// TwinCAT 3 PLC project TwinCAT_OpenFramework_Automation
// Title: TwinCAT Open Framework Automation
// Company: Oleksandr Tiutyk FOP
// Author: Oleksandr Tiutyk
// ProjectVersion: 1.0.13.0
// Description: TwinCAT.OpenFramework automation core types and device abstractions
// ProgramVersion: 3.1.4026.28
// libraries:
//   Tc2_Standard, * (Beckhoff Automation GmbH)
//   Tc2_System, * (Beckhoff Automation GmbH)
//   [TwinCAT Open Framework Core], * (Oleksandr Tiutyk FOP)
// project tree:
//   AutomationComponent/Branches/AutomationController/ AutomationController.TcPOU, AutomationControllers.TcPOU, IAutomationController.TcIO
//   AutomationComponent/Branches/AutomationController/Plugins/HMI/ HmiAutomationComponentElement.TcPOU, HMI_AUTOMATION_COMPONENT_COMMANDS.TcDUT, HMI_AUTOMATION_COMPONENT_STATUSES.TcDUT
//   AutomationComponent/Branches/AutomationController/Plugins/ IAutomationControllerPlugin.TcIO
//   AutomationComponent/Branches/ BranchAutomationComponent.TcPOU
//   AutomationComponent/Branches/Composite/ CompositeAutomationComponent.TcPOU, ICompositeAutomationComponent.TcIO
//   AutomationComponent/Branches/ChildCriticalErrorHandlingPolicies/ ChildCriticalErrorHandlingPolicies.TcPOU, CHILD_CRITICAL_ERROR_REACTION.TcDUT, IChildCriticalErrorHandlingPolicy.TcIO, IgnoreChildCriticalErrorHandlingPolicy.TcPOU, SetErrorAndContinueAfterChildCriticalErrorHandlingPolicy.TcPOU, SetErrorAndStopAfterCriticalChildErrorHandlingPolicy.TcPOU
//   AutomationComponent/Enums/ OPERATIONAL_STATE.TcDUT
//   AutomationComponent/ AutomationComponent.TcPOU, IAutomationComponent.TcIO
//   AutomationComponent/CommonSubInterfaces/ IChildAutomationComponent.TcIO, IInputLeafAutomationComponent.TcIO, IOutputLeafAutomationComponent.TcIO, IParentAutomationComponent.TcIO
//   AutomationComponent/Leafs/InputOutput/ InputOutputLeafAutomationComponent.TcPOU
//   AutomationComponent/Leafs/Input/ InputLeafAutomationComponent.TcPOU
//   AutomationComponent/Leafs/Output/ OutputLeafAutomationComponent.TcPOU
//   AutomationComponent/Leafs/ LeafAutomationComponent.TcPOU
//   AutomationRunner/ AutomationRunner.TcPOU, AUTOMATION_RUNNER_STATE.TcDUT, IAutomationRunner.TcIO
//   Internal/ CurrentNamespace.TcPOU, NamespaceExtractor.TcPOU
//   / Parameters.TcGVL
//   Simulatable/ IChildConfigurableSimulatable.TcIO, IChildSimulatable.TcIO, IConfigurableSimulatable.TcIO, ISimulatable.TcIO, SIMULATION_MODE_OVERRIDE.TcDUT
//   Version/ Global_Version.TcGVL
// (motion and I/O tree: see PLC project twincat_openframework_core)
// real-time tasks:
//   TASK PlcTask: cycle T#10ms, priority 20, ADS port 350
//   TASK TestTask: cycle T#10ms, priority 1, ADS port 351
//   TASK RunnerTestTask: cycle T#10ms, priority 2, ADS port 354
//   TASK HowToTask: cycle T#10ms, priority 22, ADS port 353
// variable links:

// ---- AutomationComponent/Branches/AutomationController/Plugins/HMI/HMI_AUTOMATION_COMPONENT_COMMANDS.TcDUT
(*
SPDX-FileCopyrightText: Â© 2026 Oleksandr Tiutyk <trofimich@gmail.com>
SPDX-License-Identifier: MIT
License: https://opensource.org/license/mit
*)

(*!
<summary>Defines command flags sent from an HMI to an automation component.</summary>
<description>
Command fields are pulsed or set by an operator/HMI interface. The element consumes and resets these flags to FALSE
within its local instance memory upon dispatching the operation.
</description>
*)

TYPE HMI_AUTOMATION_COMPONENT_COMMANDS :
STRUCT
	Enable : BOOL;
	Disable : BOOL;
	
	Reset : BOOL;	
END_STRUCT
END_TYPE

// ---- AutomationComponent/Branches/AutomationController/Plugins/HMI/HMI_AUTOMATION_COMPONENT_STATUSES.TcDUT
(*
SPDX-FileCopyrightText: Â© 2026 Oleksandr Tiutyk <trofimich@gmail.com>
SPDX-License-Identifier: MIT
License: https://opensource.org/license/mit
*)

(*!
<summary>Provides automation component operational state and diagnostics to an HMI.</summary>
<description>
Aggregates enablement, error details, and current operational state information for UI visualization.
</description>
*)

TYPE HMI_AUTOMATION_COMPONENT_STATUSES :
STRUCT
	Enabled : BOOL;

	HasError : BOOL;
	ErrorMessage : TOF_Core.ERROR_MESSAGE;
	ErrorSource : STRING(255);
	ErrorLocalTimestamp : LDATE_AND_TIME;
	ErrorUtcTimestamp : LDATE_AND_TIME;

	OperationalState : OPERATIONAL_STATE;
	OperationalStateName : STRING;
	OperationalStateReason : WSTRING(255);
END_STRUCT
END_TYPE

// ---- AutomationComponent/Branches/ChildCriticalErrorHandlingPolicies/CHILD_CRITICAL_ERROR_REACTION.TcDUT
(*
SPDX-FileCopyrightText: Â© 2026 Oleksandr Tiutyk <trofimich@gmail.com>
SPDX-License-Identifier: MIT
License: https://opensource.org/license/mit
*)

(*!
<summary>Defines reactions for handling critical errors reported by child components.</summary>
<description>
Returned by IChildCriticalErrorHandlingPolicy implementations to determine whether the parent component
should stop execution, continue running with an error state, or ignore the child failure.
</description>
*)

{attribute 'qualified_only'}
{attribute 'to_string'}
TYPE CHILD_CRITICAL_ERROR_REACTION :
(
	(*! <summary>Transition parent into error state and trigger component stop.</summary> *)
	SET_ERROR_AND_STOP,
	(*! <summary>Transition parent into error state but continue cyclic execution.</summary> *)
	SET_ERROR_AND_CONTINUE,
	(*! <summary>Ignore child error and take no action on parent component.</summary> *)
	IGNORE
);
END_TYPE

// ---- AutomationComponent/Enums/OPERATIONAL_STATE.TcDUT
(*
SPDX-FileCopyrightText: © 2026 Oleksandr Tiutyk <trofimich@gmail.com>
SPDX-License-Identifier: MIT
License: https://opensource.org/license/mit
*)

(*!
<summary>Defines the operational lifecycle states of an automation component.</summary>
*)

{attribute 'qualified_only'}
{attribute 'strict'}
{attribute 'to_string'}
TYPE OPERATIONAL_STATE :
(
	INITIALIZING := 0, (*!<description>Start state for self and children initialization.</description>*)
	WORKING,           (*!<description>Normal working mode after successful initialization.</description>*)
	(*!
	<description>
	Recoverable stopped state. Entered after Stop or critical runtime error. Reset required to return to WORKING.
	</description>
	*)
	STOPPED,
	INVALID            (*!<description>Any error occurred during initialization, final state.</description>*)
);
END_TYPE

// ---- AutomationRunner/AUTOMATION_RUNNER_STATE.TcDUT
(*
SPDX-FileCopyrightText: © 2026 Oleksandr Tiutyk <trofimich@gmail.com>
SPDX-License-Identifier: MIT
License: https://opensource.org/license/mit
*)

(*!
<summary>Defines the execution states of an automation runner.</summary>
*)

{attribute 'qualified_only'}
{attribute 'strict'}
{attribute 'to_string'}
TYPE AUTOMATION_RUNNER_STATE :
(
	INITIALIZING := 0, (*!<description>Start state, active until all components complete initialization.</description>*)
	RUNNING := 1,      (*!<description>Normal cyclic execution of automation components.</description>*)
	INVALID := 2       (*!<description>Any fatal initialization error occurred; runner execution halted.</description>*)
);
END_TYPE

// ---- Simulatable/SIMULATION_MODE_OVERRIDE.TcDUT
(*
SPDX-FileCopyrightText: Â© 2026 Oleksandr Tiutyk <trofimich@gmail.com>
SPDX-License-Identifier: MIT
License: https://opensource.org/license/mit
*)

(*!
<summary>Defines simulation mode override behavior for child components.</summary>
<description>
Allows individual child components to follow the parent's simulation state or explicitly force simulation ON or OFF.
</description>
*)

{attribute 'qualified_only'}
{attribute 'strict'}
{attribute 'to_string'}
TYPE SIMULATION_MODE_OVERRIDE :
(
	(*! <summary>Inherit simulation mode from parent component.</summary> *)
	INHERITED := 0,
	(*! <summary>Force simulation mode ON regardless of parent setting.</summary> *)
	ON,
	(*! <summary>Force simulation mode OFF regardless of parent setting.</summary> *)
	OFF
);
END_TYPE

// ---- Parameters.TcGVL
(*
SPDX-FileCopyrightText: Â© 2026 Oleksandr Tiutyk <trofimich@gmail.com>
SPDX-License-Identifier: MIT
License: https://opensource.org/license/mit
*)

(*!
<summary>Defines global configuration parameters for the automation framework.</summary>
*)

{attribute 'qualified_only'}
VAR_GLOBAL CONSTANT
	(*! <summary>Default timeout duration for component initialization phase (5 seconds).</summary> *)
	InitializationTimeout : TIME := T#5S;
END_VAR

// ---- Version/Global_Version.TcGVL
{attribute 'TcGenerated'}
{attribute 'no-analysis'}
{attribute 'linkalways'}
// This function has been automatically generated from the project information.
VAR_GLOBAL CONSTANT
	{attribute 'const_non_replaced'}
	stLibVersion_TwinCAT_Open_Framework_Automation : ST_LibVersion := (iMajor := 1, iMinor := 0, iBuild := 13, iRevision := 0, nFlags := 0, sVersion := '1.0.13.0');
END_VAR

// ---- AutomationComponent/Branches/AutomationController/IAutomationController.TcIO
(*
SPDX-FileCopyrightText: © 2026 Oleksandr Tiutyk <trofimich@gmail.com>
SPDX-License-Identifier: MIT
License: https://opensource.org/license/mit
*)

(*!
<summary>
Defines the root automation controller capable of coordinating child components and controller plugins.
</summary>
<description>Indexed Try lookups return borrowed interfaces or null and do not propagate exceptions.</description>
*)

INTERFACE IAutomationController EXTENDS IParentAutomationComponent

{attribute 'monitoring' := 'call'}
PROPERTY FINAL PluginCount : TOF_Core.INT_LENGTH
GET
END_GET
END_PROPERTY

(*!
<summary>Returns a borrowed plugin by its zero-based index.</summary>
<description>
Returns null when the entry is unavailable, the index is out of range or a nested call raises an exception.
Fatal allocation observations return null and leave the fatal latch set for the outer task boundary.
Does not transfer ownership or extend lifetime. Implementations must not propagate exceptions.
</description>
*)
METHOD TryGetPluginByIndex : IAutomationControllerPlugin
VAR_INPUT
	index : TOF_Core.INT_INDEX;
END_VAR
END_METHOD

END_INTERFACE

// ---- AutomationComponent/Branches/AutomationController/Plugins/IAutomationControllerPlugin.TcIO
(*
SPDX-FileCopyrightText: Â© 2026 Oleksandr Tiutyk <trofimich@gmail.com>
SPDX-License-Identifier: MIT
License: https://opensource.org/license/mit
*)

(*!
<summary>Defines lifecycle extension hooks for an automation controller.</summary>
<description>
Plugins intercept controller execution cycles to execute custom logic before input processing and after output
processing. Both callbacks also run while disabled in WORKING or STOPPED. Input, working or stopped,
and output phases remain gated by Enabled. Check controller.Enabled before technological actions. A before
callback may enable or disable this cycle; an after callback cannot undo completed I/O. INITIALIZING and
INVALID receive no callbacks. Arguments are borrowed for the synchronous call. Do not recursively execute
the controller.
</description>
*)

INTERFACE IAutomationControllerPlugin EXTENDS __SYSTEM.IQueryInterface

(*!
<summary>Services the controller after its enabled execution phases.</summary>
<description>
Also called while disabled in WORKING or STOPPED. Check Enabled before technological actions. The
controller is borrowed for this synchronous call; do not recursively execute it. Failures use its policy.
</description>
*)
METHOD OnAfterControllerExecute
VAR_INPUT
	controller : IAutomationController;
END_VAR
END_METHOD

(*!
<summary>Services the controller before its enabled execution phases.</summary>
<description>
Also called while disabled in WORKING or STOPPED. Check Enabled before technological actions. The
controller is borrowed for this synchronous call; do not recursively execute it. Failures use its policy.
</description>
*)
METHOD OnBeforeControllerExecute
VAR_INPUT
	controller : IAutomationController;
END_VAR
END_METHOD

END_INTERFACE

// ---- AutomationComponent/Branches/Composite/ICompositeAutomationComponent.TcIO
(*
SPDX-FileCopyrightText: © 2026 Oleksandr Tiutyk <trofimich@gmail.com>
SPDX-License-Identifier: MIT
License: https://opensource.org/license/mit
*)

(*!
<summary>
Defines a composite automation component that acts both as a parent branch and as a child leaf in the
automation hierarchy.
</summary>
*)

INTERFACE ICompositeAutomationComponent EXTENDS
	IParentAutomationComponent,
	IChildAutomationComponent,
	IInputLeafAutomationComponent,
	IOutputLeafAutomationComponent

END_INTERFACE

// ---- AutomationComponent/Branches/ChildCriticalErrorHandlingPolicies/IChildCriticalErrorHandlingPolicy.TcIO
(*
SPDX-FileCopyrightText: Â© 2026 Oleksandr Tiutyk <trofimich@gmail.com>
SPDX-License-Identifier: MIT
License: https://opensource.org/license/mit
*)

(*!
<summary>Strategy for handling critical errors reported by child components.</summary>
<description>
Determines the reaction of a parent component when one of its children enters an error state.
</description>
*)

INTERFACE IChildCriticalErrorHandlingPolicy EXTENDS TOF_Core.IObject

(*!
<summary>Evaluates child error and determines the reaction to apply to the parent component.</summary>
<param name="childWithError">Child component that reported the error.</param>
<param name="handlingObject">Parent component handling the failure.</param>
<description>Returns CHILD_CRITICAL_ERROR_REACTION indicating the action to perform.</description>
*)
METHOD HandleChildCriticalError : CHILD_CRITICAL_ERROR_REACTION
VAR_INPUT
	childWithError : IChildAutomationComponent;
	handlingObject : TOF_Core.IObject;
END_VAR
END_METHOD

END_INTERFACE

// ---- AutomationComponent/IAutomationComponent.TcIO
(*
SPDX-FileCopyrightText: © 2026 Oleksandr Tiutyk <trofimich@gmail.com>
SPDX-License-Identifier: MIT
License: https://opensource.org/license/mit
*)

(*!
<summary>Defines an automation component's lifecycle, diagnostics and event delivery capabilities.</summary>
<description>
Every component can receive both bubbling and broadcast events, including roots and leaves. Delivery and
forwarding do not depend on Enabled or operational state; each recipient decides whether to react in its
current state. Being disabled or stopped does not itself stop propagation. Terminal nodes receive an event
without forwarding it; delivery uses the synchronous borrowed IEventDispatcher contract.
</description>
*)

INTERFACE IAutomationComponent EXTENDS
	TOF_Core.INamed,
	TOF_Core.IErrorProvider,
	TOF_Core.IExecutable,
	TOF_Core.IEventDispatcher

(*!
<summary>Disables cyclic execution and invokes disable hooks.</summary>
<description>
Branches also disable their children. Exceptions from disable hooks propagate to the caller without rolling
back prior effects.
</description>
*)
METHOD FINAL Disable
END_METHOD

(*!
<summary>Enables cyclic execution and invokes enable hooks.</summary>
<description>
Enabling does not automatically reset a STOPPED component. Components stopped while disabled or disabled
while stopped remain STOPPED after Enable until explicitly Reset. Child enablement also enables disabled
parents with includeChildren := FALSE.
</description>
<param name="includeChildren">When TRUE on a branch, recursively enables child components.</param>
*)
METHOD FINAL Enable
VAR_INPUT
	includeChildren : BOOL := TRUE;
END_VAR
END_METHOD

{attribute 'monitoring' := 'call'}
PROPERTY Enabled : BOOL
GET
END_GET
END_PROPERTY

METHOD FINAL GetEffectiveExceptionHandlingPolicy : TOF_Core.IExceptionHandlingPolicy
END_METHOD

(*!
<summary>Sets the maximum wait for pending initialization.</summary>
<description>
T#0S selects Parameters.InitializationTimeout immediately upon assignment, so the getter always returns the
active non-zero duration. During initialization, a branch expands its effective initialization timeout to at
least the maximum InitializationTimeout of its children.
</description>
*)
{attribute 'monitoring' := 'call'}
PROPERTY InitializationTimeout : TIME
GET
END_GET
SET
END_SET
END_PROPERTY

(*!
<summary>Advances initialization after validating mandatory dependencies.</summary>
<description>
Child components require a live constructor-bound parent. Missing required dependencies fail before
initialization hooks. FALSE reports pending work or failure; INVALID never reports TRUE. Caught failures
record a copied critical error in terminal INVALID. Already initialized or stopped components report TRUE.
Completed callback effects are not rolled back.
Only a pending call evaluates the timeout. Completion on the deadline cycle succeeds.
</description>
*)
METHOD Initialize : BOOL
END_METHOD

{attribute 'monitoring' := 'call'}
PROPERTY FINAL OperationalState : OPERATIONAL_STATE
GET
END_GET
END_PROPERTY

{attribute 'monitoring' := 'call'}
PROPERTY FINAL OperationalStateReason : REFERENCE TO WSTRING(255)
GET
END_GET
END_PROPERTY

(*!
<summary>Attempts to recover an enabled stopped component to WORKING.</summary>
<description>
Served only while Enabled and in OPERATIONAL_STATE.STOPPED. Clears the execution error before reset hooks.
A failure in the component's own reset hook (OnReset, OnBeforeChildrenReset or OnAfterChildrenReset) always
leaves the component in OPERATIONAL_STATE.STOPPED with a copied CRITICAL error without consulting the
exception handling policy.
</description>
*)
METHOD Reset
END_METHOD

(*!
<summary>Transitions a WORKING component to OPERATIONAL_STATE.STOPPED.</summary>
<description>
Transitions a WORKING component (and, for branches, all WORKING children) to OPERATIONAL_STATE.STOPPED
regardless of Enabled.
</description>
<param name="reason">Descriptive reason stored in OperationalStateReason.</param>
*)
METHOD FINAL Stop
VAR_INPUT
	reason : WSTRING(255) := "External stop";
END_VAR
END_METHOD

END_INTERFACE

// ---- AutomationComponent/CommonSubInterfaces/IChildAutomationComponent.TcIO
(*
SPDX-FileCopyrightText: © 2026 Oleksandr Tiutyk <trofimich@gmail.com>
SPDX-License-Identifier: MIT
License: https://opensource.org/license/mit
*)

(*!
<summary>Describes an automation component with a parent in the component hierarchy.</summary>
<description>
Both event delivery directions are inherited from IAutomationComponent; bubbling can continue through Parent.
</description>
*)

INTERFACE IChildAutomationComponent EXTENDS IAutomationComponent

{attribute 'monitoring' := 'call'}
PROPERTY Parent : IParentAutomationComponent
GET
END_GET
END_PROPERTY

END_INTERFACE

// ---- AutomationComponent/CommonSubInterfaces/IInputLeafAutomationComponent.TcIO
(*
SPDX-FileCopyrightText: Â© 2026 Oleksandr Tiutyk <trofimich@gmail.com>
SPDX-License-Identifier: MIT
License: https://opensource.org/license/mit
*)

(*!
<summary>Represents a leaf automation component that performs cyclic input processing.</summary>
<description>
Invoked during the input phase of the component tree cycle to read physical inputs or update state.
</description>
*)

INTERFACE IInputLeafAutomationComponent EXTENDS IChildAutomationComponent

(*!
<summary>Performs cyclic reading and processing of input data.</summary>
*)
METHOD ProcessInput
END_METHOD

END_INTERFACE

// ---- AutomationComponent/CommonSubInterfaces/IOutputLeafAutomationComponent.TcIO
(*
SPDX-FileCopyrightText: Â© 2026 Oleksandr Tiutyk <trofimich@gmail.com>
SPDX-License-Identifier: MIT
License: https://opensource.org/license/mit
*)

(*!
<summary>Represents a leaf automation component that performs cyclic output processing.</summary>
<description>
Invoked during the output phase of the component tree cycle to write physical outputs or command actuators.
</description>
*)

INTERFACE IOutputLeafAutomationComponent EXTENDS IChildAutomationComponent

(*!
<summary>Performs cyclic writing and processing of output data.</summary>
*)
METHOD ProcessOutput
END_METHOD

END_INTERFACE

// ---- AutomationComponent/CommonSubInterfaces/IParentAutomationComponent.TcIO
(*
SPDX-FileCopyrightText: © 2026 Oleksandr Tiutyk <trofimich@gmail.com>
SPDX-License-Identifier: MIT
License: https://opensource.org/license/mit
*)

(*!
<summary>
Describes an automation component that exposes children, dispatches broadcasts and provides action
permissions.
</summary>
<description>
Permission requests are evaluated locally and then through parents; the first rejection ends evaluation.
Each child in the execution hierarchy occupies one slot and identifies its containing branch as Parent.
Other components may borrow the same child independently of this hierarchy.
Indexed Try lookups return borrowed interfaces or null and do not propagate exceptions.
</description>
*)
INTERFACE IParentAutomationComponent EXTENDS IAutomationComponent, TOF_Core.IActionPermissionProvider

{attribute 'monitoring' := 'call'}
PROPERTY FINAL ActionPermissionPolicy : TOF_Core.IActionPermissionPolicy
GET
END_GET
SET
END_SET
END_PROPERTY

{attribute 'monitoring' := 'call'}
PROPERTY ChildCount : TOF_Core.INT_LENGTH
GET
END_GET
END_PROPERTY

{attribute 'monitoring' := 'call'}
PROPERTY FINAL ChildCriticalErrorHandlingPolicy : IChildCriticalErrorHandlingPolicy
GET
END_GET
SET
END_SET
END_PROPERTY

METHOD GetEffectiveChildCriticalErrorHandlingPolicy : IChildCriticalErrorHandlingPolicy
END_METHOD

(*!
<summary>Requests permission from this level and its parents, stopping at the first rejection.</summary>
<description>
A missing policy permits its level; the request succeeds only if no level rejects it. The
IActionPermissionProvider contract applies: live non-null inputs, synchronous borrowing, current rejectReason
on FALSE, ignored rejectReason on TRUE, and propagation of evaluation exceptions.
</description>
*)

METHOD RequestActionPermission : BOOL
VAR_INPUT
	actionDescriptor : TOF_Core.INamed;
	requestingObject : TOF_Core.IObject;
END_VAR
VAR_IN_OUT
	rejectReason : WSTRING(255);
END_VAR
END_METHOD

(*!
<summary>Returns a borrowed child by its zero-based index.</summary>
<description>
Returns null when the entry is unavailable, the index is out of range or a nested call raises an exception.
Fatal allocation observations return null and leave the fatal latch set for the outer task boundary.
Does not transfer ownership or extend lifetime. Implementations must not propagate exceptions.
</description>
*)
METHOD TryGetChildByIndex : IChildAutomationComponent
VAR_INPUT
	index : TOF_Core.INT_INDEX;
END_VAR
END_METHOD

END_INTERFACE

// ---- AutomationRunner/IAutomationRunner.TcIO
(*
SPDX-FileCopyrightText: Â© 2026 Oleksandr Tiutyk <trofimich@gmail.com>
SPDX-License-Identifier: MIT
License: https://opensource.org/license/mit
*)

(*!
<summary>Provides cyclic execution and initialization state of automation components.</summary>
<description>
Execute advances the fixed sequence of roots bound at construction. State and StateName describe runner initialization.
</description>
*)

INTERFACE IAutomationRunner EXTENDS TOF_Core.IObject

(*!
<summary>Initializes and advances cyclic execution of the registered components.</summary>
<description>
Validates the bound roots before the first root initialization. An empty array, null slot or repeated instance
makes the runner INVALID. After initialization succeeds, subsequent calls execute roots in array order.
Call from the outer task boundary. Nested runner execution is unsupported because cleanup covers the calling task.
Call at the task boundary outside handlers that swallow terminal allocation failures.
</description>
*)
METHOD FINAL Execute
END_METHOD

(*!
<summary>Gets current initialization and operational state of the runner.</summary>
*)
{attribute 'monitoring' := 'call'}
PROPERTY FINAL State : AUTOMATION_RUNNER_STATE
GET
END_GET
END_PROPERTY

(*!
<summary>Gets string representation of current runner state.</summary>
*)
{attribute 'monitoring' := 'call'}
PROPERTY StateName : STRING
GET
END_GET
END_PROPERTY

END_INTERFACE

// ---- Simulatable/IChildConfigurableSimulatable.TcIO
(*
SPDX-FileCopyrightText: Â© 2026 Oleksandr Tiutyk <trofimich@gmail.com>
SPDX-License-Identifier: MIT
License: https://opensource.org/license/mit
*)

(*!
<summary>Represents a child automation component whose simulation override can be configured.</summary>
*)

INTERFACE IChildConfigurableSimulatable EXTENDS IChildSimulatable

(*!
<summary>Configures the simulation mode override setting for this child component.</summary>
<param name="value">Override setting (INHERITED, ON, or OFF).</param>
*)
METHOD SetSimulationModeOverride
VAR_INPUT
	value : SIMULATION_MODE_OVERRIDE;
END_VAR
END_METHOD

END_INTERFACE

// ---- Simulatable/IChildSimulatable.TcIO
(*
SPDX-FileCopyrightText: Â© 2026 Oleksandr Tiutyk <trofimich@gmail.com>
SPDX-License-Identifier: MIT
License: https://opensource.org/license/mit
*)

(*!
<summary>Represents a child automation component with an overridable simulation mode.</summary>
*)

INTERFACE IChildSimulatable EXTENDS ISimulatable

(*!
<summary>Gets the simulation mode override setting for this child component.</summary>
*)
{attribute 'monitoring' := 'call'}
PROPERTY SimulationModeOverride : SIMULATION_MODE_OVERRIDE
GET
END_GET
END_PROPERTY

END_INTERFACE

// ---- Simulatable/IConfigurableSimulatable.TcIO
(*
SPDX-FileCopyrightText: Â© 2026 Oleksandr Tiutyk <trofimich@gmail.com>
SPDX-License-Identifier: MIT
License: https://opensource.org/license/mit
*)

(*!
<summary>Represents an automation component with configurable simulation mode.</summary>
*)

INTERFACE IConfigurableSimulatable EXTENDS ISimulatable

(*!
<summary>Sets whether simulation mode is enabled for the component.</summary>
<param name="value">TRUE to enable simulation mode, FALSE to use physical hardware.</param>
*)
METHOD SetSimulationMode
VAR_INPUT
	value : BOOL;
END_VAR
END_METHOD

END_INTERFACE

// ---- Simulatable/ISimulatable.TcIO
(*
SPDX-FileCopyrightText: Â© 2026 Oleksandr Tiutyk <trofimich@gmail.com>
SPDX-License-Identifier: MIT
License: https://opensource.org/license/mit
*)

(*!
<summary>Represents an automation component capable of operating in simulation mode.</summary>
<description>
Provides read access to the active simulation mode status.
</description>
*)

INTERFACE ISimulatable EXTENDS TOF_Core.IObject

(*!
<summary>Gets whether simulation mode is currently active.</summary>
*)
{attribute 'monitoring' := 'call'}
PROPERTY SimulationMode : BOOL
GET
END_GET
END_PROPERTY

END_INTERFACE

// ---- AutomationComponent/Branches/AutomationController/AutomationController.TcPOU
(*
SPDX-FileCopyrightText: © 2026 Oleksandr Tiutyk <trofimich@gmail.com>
SPDX-License-Identifier: MIT
License: https://opensource.org/license/mit
*)

(*!
<summary>Coordinates the root of an automation component tree and its controller plugins.</summary>
<description>
Use the inherited BroadcastEvent to deliver events to this controller and its descendants. The inherited
BubbleEvent receives events at the root without forwarding them further. Both operations use synchronous
borrowed delivery and do not transfer event ownership. Indexed Try lookups return borrowed interfaces or null
and do not propagate exceptions. Fatal allocation observations return null without clearing the latch.
A state transition during output processing skips remaining outputs and the after-output hook.
Completed writes remain effective. A pass started in STOPPED proceeds while the branch stays in that state.
Plugin callbacks run in WORKING and STOPPED even while disabled, independently of enabled I/O and working
or stopped hooks. INITIALIZING and INVALID receive no cycle callbacks.
</description>
*)

FUNCTION_BLOCK ABSTRACT AutomationController 
VAR_GENERIC CONSTANT
	{attribute 'hide'} 
    _ChildCount : TOF_Core.INT_LENGTH := 0;
END_VAR
EXTENDS BranchAutomationComponent IMPLEMENTS IAutomationController
VAR
	{attribute 'hide'} 
	_Plugins : POINTER TO IAutomationControllerPlugin;
	{attribute 'hide'} 
    _PluginCount : TOF_Core.INT_LENGTH := 0;
END_VAR

METHOD PROTECTED AssignPlugins
VAR_IN_OUT CONSTANT
	plugins : ARRAY [*] OF IAutomationControllerPlugin;
END_VAR
IF __ISVALIDREF(plugins) THEN
	_Plugins := plugins;
	_PluginCount := TO_INT(1 + UPPER_BOUND(plugins, 1) - LOWER_BOUND(plugins, 1));
END_IF
END_METHOD

{attribute 'monitoring' := 'call'}
PROPERTY FINAL ChildCount : TOF_Core.INT_LENGTH
GET
ChildCount := _ChildCount;
END_GET
END_PROPERTY

{attribute 'monitoring' := 'call'}
PROPERTY ABSTRACT Children : REFERENCE TO ARRAY [0.._ChildCount - 1] OF IChildAutomationComponent
GET
END_GET
END_PROPERTY

(*!
<summary>Processes child outputs after the working or stopped phase.</summary>
<description>
Execute checks Enabled before entering this phase. An enabled controller processes outputs in both WORKING
and STOPPED.
A state transition during output processing skips remaining outputs and the after-output hook.
Completed writes remain effective. A pass started in STOPPED proceeds while the branch stays in that state.
OnCycleEnd can still dispatch plugin callbacks when this phase is skipped.
</description>
*)
METHOD PROTECTED FINAL OnAfterExecute
VAR
	entryRevision : UDINT;
	exceptionCode : __SYSTEM.ExceptionCode;
	exception : TOF_Core.IException;	
	exceptionReaction : TOF_Core.EXCEPTION_REACTION;

	childCriticalErrorReaction : CHILD_CRITICAL_ERROR_REACTION;

	i : TOF_Core.INT_INDEX;
	
	child : IChildAutomationComponent;
	
	outputDevice : IOutputLeafAutomationComponent;
END_VAR
entryRevision := _OperationalStateRevision;

__TRY
	OnBeforeChildrenProcessOutput();
__CATCH(exceptionCode)		
	exception := TOF_Core.ExceptionManager.GetLastException(
		exceptionCode := exceptionCode,
		catchPointNamespaceName := NamespaceName,
		catchPointPOUName := __POUNAME(),
		catchPointPosition := __POSITION()
	);
					
	exceptionReaction := OnHandleException(exception := exception, failedMethodName := 'OnBeforeChildrenProcessOutput');

	ProcessException(
		exception := exception,
		exceptionReaction := exceptionReaction,
		exceptionSourceHint := "OnBeforeChildrenProcessOutput error"
	);
__ENDTRY

FOR i := 0 TO ChildCount - 1 DO
	IF _OperationalStateRevision <> entryRevision THEN
		RETURN;
	END_IF

	child := TryGetChildByIndex(index := i);
	
	IF child = 0 OR_ELSE NOT child.Enabled OR_ELSE NOT __QUERYINTERFACE(child, outputDevice) THEN
		CONTINUE;
	END_IF

	IF _OperationalStateRevision <> entryRevision THEN
		RETURN;
	END_IF

	outputDevice.ProcessOutput(); 
	
	IF outputDevice.HasError AND_THEN outputDevice.Error.Severity = TOF_Core.ERROR_SEVERITY.CRITICAL THEN
		childCriticalErrorReaction := HandleChildCriticalError(childWithError := outputDevice);
		
		ProcessChildError(
			childError := outputDevice.Error,
			childErrorReaction := childCriticalErrorReaction,
			childErrorSourceHint := TOF_Core.WideStrings.Concat255(
				"Child[",
				TO_WSTRING(i),
				"](",
				outputDevice.Name,
				").ProcessOutput error"
			)
		);
	END_IF
END_FOR

IF _OperationalStateRevision <> entryRevision THEN
	RETURN;
END_IF

__TRY
	OnAfterChildrenProcessOutput();
__CATCH(exceptionCode)		
	exception := TOF_Core.ExceptionManager.GetLastException(
		exceptionCode := exceptionCode,
		catchPointNamespaceName := NamespaceName,
		catchPointPOUName := __POUNAME(),
		catchPointPosition := __POSITION()
	);
					
	exceptionReaction := OnHandleException(exception := exception, failedMethodName := 'OnAfterChildrenProcessOutput');

	ProcessException(
		exception := exception,
		exceptionReaction := exceptionReaction,
		exceptionSourceHint := "OnAfterChildrenProcessOutput error"
	);
__ENDTRY
END_METHOD

(*!
<summary>Processes child inputs before the working or stopped phase.</summary>
<description>
Execute checks Enabled after OnCycleStart before entering this phase. An enabled controller processes
inputs in both WORKING and STOPPED.
While the branch remains enabled, a transition to STOPPED continues the input pass through the remaining
enabled input children and the after-input hook. Input callbacks must support execution in STOPPED.
</description>
*)
METHOD PROTECTED FINAL OnBeforeExecute
VAR
	exceptionCode : __SYSTEM.ExceptionCode;
	exception : TOF_Core.IException;	
	exceptionReaction : TOF_Core.EXCEPTION_REACTION;

	childCriticalErrorReaction : CHILD_CRITICAL_ERROR_REACTION;

	i : TOF_Core.INT_INDEX;

	child : IChildAutomationComponent;
	
	inputDevice : IInputLeafAutomationComponent;
END_VAR
__TRY
	OnBeforeChildrenProcessInput();
__CATCH(exceptionCode)		
	exception := TOF_Core.ExceptionManager.GetLastException(
		exceptionCode := exceptionCode,
		catchPointNamespaceName := NamespaceName,
		catchPointPOUName := __POUNAME(),
		catchPointPosition := __POSITION()
	);
					
	exceptionReaction := OnHandleException(exception := exception, failedMethodName := 'OnBeforeChildrenProcessInput');

	ProcessException(
		exception := exception,
		exceptionReaction := exceptionReaction,
		exceptionSourceHint := "OnBeforeChildrenProcessInput error"
	);
__ENDTRY

FOR i := 0 TO ChildCount - 1 DO
	child := TryGetChildByIndex(index := i);

	IF child = 0 OR_ELSE NOT child.Enabled OR_ELSE NOT __QUERYINTERFACE(child, inputDevice) THEN
		CONTINUE;
	END_IF

	inputDevice.ProcessInput(); 

	IF inputDevice.HasError AND_THEN inputDevice.Error.Severity = TOF_Core.ERROR_SEVERITY.CRITICAL THEN
		childCriticalErrorReaction := HandleChildCriticalError(childWithError := inputDevice);
		
		ProcessChildError(
			childError := inputDevice.Error,
			childErrorReaction := childCriticalErrorReaction,
			childErrorSourceHint := TOF_Core.WideStrings.Concat255(
				"Child[",
				TO_WSTRING(i),
				"](",
				inputDevice.Name,
				").ProcessInput error"
			)
		);
	END_IF	
END_FOR

__TRY
	OnAfterChildrenProcessInput();
__CATCH(exceptionCode)		
	exception := TOF_Core.ExceptionManager.GetLastException(
		exceptionCode := exceptionCode,
		catchPointNamespaceName := NamespaceName,
		catchPointPOUName := __POUNAME(),
		catchPointPosition := __POSITION()
	);
					
	exceptionReaction := OnHandleException(exception := exception, failedMethodName := 'OnAfterChildrenProcessInput');

	ProcessException(
		exception := exception,
		exceptionReaction := exceptionReaction,
		exceptionSourceHint := "OnAfterChildrenProcessInput error"
	);
__ENDTRY
END_METHOD

{attribute 'monitoring' := 'call'}
PROPERTY FINAL PluginCount : TOF_Core.INT_LENGTH
GET
PluginCount := _PluginCount;
END_GET
END_PROPERTY

(*!
<summary>Returns a borrowed child by its zero-based index.</summary>
<description>
Returns null when the entry is unavailable, the index is out of range or a nested call raises an exception.
Fatal allocation observations before or after the storage getter return null and preserve the latch for
the outer task boundary. Does not transfer ownership or extend lifetime. Getter exceptions are contained.
</description>
*)
METHOD FINAL TryGetChildByIndex : IChildAutomationComponent
VAR_INPUT
	index : TOF_Core.INT_INDEX;
END_VAR
VAR
	childStorage : REFERENCE TO ARRAY [0.._ChildCount - 1] OF IChildAutomationComponent;
END_VAR
__TRY
	IF TOF_Core.DynamicMemoryManager.HasAllocationFailed OR_ELSE index < 0 OR_ELSE index >= _ChildCount THEN
		RETURN;
	END_IF

	childStorage REF= Children;

	IF NOT TOF_Core.DynamicMemoryManager.HasAllocationFailed AND_THEN __ISVALIDREF(childStorage) THEN
		TryGetChildByIndex := childStorage[index];
	END_IF
__CATCH
	TryGetChildByIndex := 0;
__ENDTRY

IF TOF_Core.DynamicMemoryManager.HasAllocationFailed THEN
	TryGetChildByIndex := 0;
END_IF
END_METHOD

(*!
<summary>Returns a borrowed plugin by its zero-based index.</summary>
<description>
Returns null when the entry is unavailable, the index is out of range or a nested call raises an exception.
Fatal allocation observations return null and preserve the latch for the task boundary.
Does not transfer ownership or extend lifetime; no exception may escape.
</description>
*)
METHOD FINAL TryGetPluginByIndex : IAutomationControllerPlugin
VAR_INPUT
	index : TOF_Core.INT_INDEX;
END_VAR
__TRY
	IF TOF_Core.DynamicMemoryManager.HasAllocationFailed THEN
		RETURN;
	END_IF

	IF _Plugins <> 0 AND_THEN index >= 0 AND_THEN index < _PluginCount THEN
		TryGetPluginByIndex := _Plugins[index];
	END_IF
__CATCH
	TryGetPluginByIndex := 0;
__ENDTRY

IF TOF_Core.DynamicMemoryManager.HasAllocationFailed THEN
	TryGetPluginByIndex := 0;
END_IF
END_METHOD

METHOD PROTECTED FINAL Validate
VAR
END_VAR
IF ChildCount > 0 AND_THEN NOT __ISVALIDREF(Children) THEN
	TOF_Core.Exceptions.ThrowDataMemberNotSpecified(
		sourceNamespaceName := NamespaceName,
		sourceClassName := ClassName,
		sourcePOUName := __POUNAME(),
		sourcePosition := __POSITION(),
		dataMemberName := 'Children'
	);
END_IF
END_METHOD

(*!
<summary>Dispatches OnBeforeControllerExecute to controller plugins before child input processing.</summary>
<description>
Plugins receive this callback in WORKING and STOPPED, including while disabled. Changes to Enabled affect
input processing in this call. Plugins must check Enabled before performing technological actions.
Plugin failures follow the controller exception policy. Completed callback effects are retained.
</description>
*)
METHOD PROTECTED FINAL OnCycleStart
VAR
	i : TOF_Core.INT_INDEX;
	plugin : IAutomationControllerPlugin;

	exceptionCode : __SYSTEM.ExceptionCode;
	exception : TOF_Core.IException;
	exceptionReaction : TOF_Core.EXCEPTION_REACTION;
END_VAR
FOR i := 0 TO PluginCount - 1 DO
	plugin := TryGetPluginByIndex(index := i);
	
	IF plugin <> 0 THEN
		__TRY
			plugin.OnBeforeControllerExecute(controller := THIS^);
		__CATCH(exceptionCode)		
			exception := TOF_Core.ExceptionManager.GetLastException(
				exceptionCode := exceptionCode,
				catchPointNamespaceName := NamespaceName,
				catchPointPOUName := __POUNAME(),
				catchPointPosition := __POSITION()
			);
							
			exceptionReaction := OnHandleException(
				exception := exception,
				failedMethodName := TOF_Core.Strings.Concat255('plugin[', TO_STRING(i), '].OnBeforeControllerExecute')
			);
		
			ProcessException(
				exception := exception,
				exceptionReaction := exceptionReaction,
				exceptionSourceHint := TOF_Core.WideStrings.Concat255("plugin[", TO_WSTRING(i), "].OnBeforeControllerExecute error")
			);
		__ENDTRY		
	END_IF
END_FOR
END_METHOD

(*!
<summary>Dispatches OnAfterControllerExecute so plugins can observe the resulting controller state.</summary>
<description>
Plugins receive this callback even when the enabled phases were skipped. An escaping failure can end Execute
before dispatch. Plugins must check Enabled before performing technological actions. Plugin failures follow
the controller exception policy. Completed callback effects are retained.
</description>
*)
METHOD PROTECTED FINAL OnCycleEnd
VAR
	i : TOF_Core.INT_INDEX;
	plugin : IAutomationControllerPlugin;

	exceptionCode : __SYSTEM.ExceptionCode;
	exception : TOF_Core.IException;
	exceptionReaction : TOF_Core.EXCEPTION_REACTION;
END_VAR
FOR i := 0 TO PluginCount - 1 DO
	plugin := TryGetPluginByIndex(index := i);
	
	IF plugin <> 0 THEN
		__TRY
			plugin.OnAfterControllerExecute(controller := THIS^);
		__CATCH(exceptionCode)		
			exception := TOF_Core.ExceptionManager.GetLastException(
				exceptionCode := exceptionCode,
				catchPointNamespaceName := NamespaceName,
				catchPointPOUName := __POUNAME(),
				catchPointPosition := __POSITION()
			);
							
			exceptionReaction := OnHandleException(
				exception := exception,
				failedMethodName := TOF_Core.Strings.Concat255('plugin[', TO_STRING(i), '].OnAfterControllerExecute')
			);
		
			ProcessException(
				exception := exception,
				exceptionReaction := exceptionReaction,
				exceptionSourceHint := TOF_Core.WideStrings.Concat255("plugin[", TO_WSTRING(i), "].OnAfterControllerExecute error")
			);
		__ENDTRY		
	END_IF
END_FOR
END_METHOD

END_FUNCTION_BLOCK

// ---- AutomationComponent/Branches/BranchAutomationComponent.TcPOU
(*
SPDX-FileCopyrightText: © 2026 Oleksandr Tiutyk <trofimich@gmail.com>
SPDX-License-Identifier: MIT
License: https://opensource.org/license/mit
*)

(*!
<summary>
Base automation component that coordinates children and routes requests through the component hierarchy.
</summary>
<description>
Action permissions are checked locally and then through parents, stopping at the first rejection. A missing
local policy permits that level; permission is granted only if no level rejects the request. Indexed Try
lookups return borrowed interfaces or null and do not propagate exceptions. Initialization validates required
dependencies before hooks. Each fixed child slot must identify a distinct child whose Parent is this branch.
Cycle-service hooks remain available while disabled in WORKING or STOPPED;
state changes end obsolete child phases. Use one owner task without recursive Execute.
</description>
*)

FUNCTION_BLOCK ABSTRACT BranchAutomationComponent EXTENDS AutomationComponent IMPLEMENTS IParentAutomationComponent
VAR
	{attribute 'hide'} 
	_ActionPermissionPolicy : TOF_Core.IActionPermissionPolicy;
	
	{attribute 'hide'} 
	_ChildCriticalErrorHandlingPolicy : IChildCriticalErrorHandlingPolicy;

	_ChildHierarchyValidated : BOOL;
END_VAR

{attribute 'monitoring' := 'call'}
PROPERTY FINAL ActionPermissionPolicy : TOF_Core.IActionPermissionPolicy
GET
ActionPermissionPolicy := _ActionPermissionPolicy;
END_GET
SET
_ActionPermissionPolicy := ActionPermissionPolicy;
END_SET
END_PROPERTY

METHOD FINAL BroadcastEvent
VAR_INPUT
	event : TOF_Core.IEvent;
END_VAR
VAR
	stopPropagation : BOOL;
	
	i : TOF_Core.INT_INDEX;
	
	child : IChildAutomationComponent;
	childAsBroadcastEventDispatcher : TOF_Core.IBroadcastEventDispatcher;
END_VAR
OnEventReceived(event := event, stopPropagation => stopPropagation);

IF stopPropagation THEN
	RETURN;
END_IF

FOR i := 0 TO ChildCount - 1 DO
	child := TryGetChildByIndex(index := i);
	
	IF child = 0 OR_ELSE NOT __QUERYINTERFACE(child, childAsBroadcastEventDispatcher) THEN
		CONTINUE;
	END_IF
	
	childAsBroadcastEventDispatcher.BroadcastEvent(event := event);
END_FOR
END_METHOD

{attribute 'monitoring' := 'call'}
PROPERTY ABSTRACT ChildCount : TOF_Core.INT_LENGTH
GET
END_GET
END_PROPERTY

{attribute 'monitoring' := 'call'}
PROPERTY FINAL ChildCriticalErrorHandlingPolicy : IChildCriticalErrorHandlingPolicy
GET
ChildCriticalErrorHandlingPolicy := _ChildCriticalErrorHandlingPolicy;
END_GET
SET
_ChildCriticalErrorHandlingPolicy := ChildCriticalErrorHandlingPolicy;
END_SET
END_PROPERTY

(*!
<summary>Disables the branch, its children and invokes disable hooks.</summary>
<description>
Hook or child exceptions propagate to the caller without rolling back already disabled children.
</description>
*)
METHOD FINAL Disable
VAR
	i : INT;
	
	child : IChildAutomationComponent;

	exceptionCode : __SYSTEM.ExceptionCode;
END_VAR
VAR_INST
	disabling : BOOL;
END_VAR
IF NOT _Enabled OR_ELSE disabling THEN
	RETURN;
END_IF

disabling := TRUE;

__TRY
	OnBeforeChildrenDisable();
	
	FOR i := 0 TO ChildCount - 1 DO
		child := TryGetChildByIndex(index := i);
		
		IF child <> 0 THEN
			child.Disable();
		END_IF
	END_FOR
	
	OnAfterChildrenDisable();
	
	_Enabled := FALSE;
	
	disabling := FALSE;	
__CATCH(exceptionCode)
	disabling := FALSE;
	
	TOF_Core.ExceptionManager.ReThrowLastException(
		exceptionCode := exceptionCode,
		catchPointNamespaceName := NamespaceName,
		catchPointPOUName := __POUNAME(),
		catchPointPosition := __POSITION()
	);
__ENDTRY
END_METHOD

(*!
<summary>Advances stopped children while the branch remains enabled and stopped.</summary>
<description>
OnBeforeChildrenStopped may call Reset. A state or enablement change ends this phase before remaining
children or the after-stopped hook. Completed effects remain. Hook failures are logged; other failures may escape.
</description>
*)
METHOD PRIVATE FINAL doStop
VAR
	exceptionCode : __SYSTEM.ExceptionCode;
	exception : TOF_Core.IException;	
	exceptionReaction : TOF_Core.EXCEPTION_REACTION;

	i : INT;
	
	child : IChildAutomationComponent;
END_VAR
__TRY
	OnBeforeChildrenStopped();
__CATCH(exceptionCode)
	exception := TOF_Core.ExceptionManager.GetLastException(
		exceptionCode := exceptionCode,
		catchPointNamespaceName := NamespaceName,
		catchPointPOUName := __POUNAME(),
		catchPointPosition := __POSITION()
	);	

	exceptionReaction := OnHandleException(exception := exception, failedMethodName := 'OnBeforeChildrenStopped');

	TOF_Core.LogManager.TryLogException(
		exception := exception,
		severity := GetErrorSeverityByExceptionReaction(exceptionReaction := exceptionReaction),
		topic1 := "AutomationComponent",
		topic2 := "AutomationComponent.OnBeforeChildrenStopped"
	);
__ENDTRY	

IF NOT Enabled OR_ELSE _OperationalState <> OPERATIONAL_STATE.STOPPED THEN
	RETURN;
END_IF

FOR i := 0 TO ChildCount - 1 DO
	child := TryGetChildByIndex(index := i);
	
	IF child = 0 OR_ELSE NOT child.Enabled THEN
		CONTINUE;
	END_IF
	
	CASE child.OperationalState OF
		OPERATIONAL_STATE.WORKING:			
			child.Stop(reason := TOF_Core.WideStrings.Concat255("Parent device (", Name, ") stopped"));
		
		OPERATIONAL_STATE.STOPPED:
			child.Execute();
	END_CASE

	IF NOT Enabled OR_ELSE _OperationalState <> OPERATIONAL_STATE.STOPPED THEN
		RETURN;
	END_IF
END_FOR

__TRY
	OnAfterChildrenStopped();
__CATCH(exceptionCode)
	exception := TOF_Core.ExceptionManager.GetLastException(
		exceptionCode := exceptionCode,
		catchPointNamespaceName := NamespaceName,
		catchPointPOUName := __POUNAME(),
		catchPointPosition := __POSITION()
	);	

	exceptionReaction := OnHandleException(exception := exception, failedMethodName := 'OnAfterChildrenStopped');

	TOF_Core.LogManager.TryLogException(
		exception := exception,
		severity := GetErrorSeverityByExceptionReaction(exceptionReaction := exceptionReaction),
		topic1 := "AutomationComponent",
		topic2 := "AutomationComponent.OnAfterChildrenStopped"
	);
__ENDTRY
END_METHOD

(*!
<summary>Advances children according to the selected critical-error reaction.</summary>
<description>
Ignore and continue preserve traversal of later children and the after-working hook. Stop ends traversal.
A non-critical error copied from a faulted child under SET_ERROR_AND_CONTINUE is retained without calling
OnRecover while any enabled child still holds a critical error handled with continue. An exception raised by
OnRecover always records a copied CRITICAL error and stops the branch without consulting
ExceptionHandlingPolicy. State or enablement changes end the obsolete phase; completed effects remain.
</description>
*)
METHOD PRIVATE doWork
VAR
	exceptionCode : __SYSTEM.ExceptionCode;
	exception : TOF_Core.IException;	
	exceptionReaction : TOF_Core.EXCEPTION_REACTION;

	childCriticalErrorReaction : CHILD_CRITICAL_ERROR_REACTION;

	i : INT;
	
	child : IChildAutomationComponent;
END_VAR
// automatic non-critical error recovering
IF _OperationalState = OPERATIONAL_STATE.WORKING
	AND_THEN HasError
	AND_THEN _Error.Severity <> TOF_Core.ERROR_SEVERITY.CRITICAL
	AND_THEN NOT hasActiveChildCriticalError()
THEN
	_Error.Clear();
	
	__TRY
		OnRecover();
	__CATCH(exceptionCode)		
		exception := TOF_Core.ExceptionManager.GetLastException(
			exceptionCode := exceptionCode,
			catchPointNamespaceName := NamespaceName,
			catchPointPOUName := __POUNAME(),
			catchPointPosition := __POSITION()
		);

		// An OnRecover failure always stops the branch with a critical error without consulting the policy.
		ProcessException(
			exception := exception,
			exceptionReaction := TOF_Core.EXCEPTION_REACTION.SET_ERROR_AND_STOP,
			exceptionSourceHint := "OnRecover error"
		);

		RETURN;
	__ENDTRY
END_IF

IF NOT Enabled OR_ELSE _OperationalState <> OPERATIONAL_STATE.WORKING THEN
	RETURN;
END_IF

__TRY
	OnBeforeChildrenWorking();
__CATCH(exceptionCode)
	exception := TOF_Core.ExceptionManager.GetLastException(
		exceptionCode := exceptionCode,
		catchPointNamespaceName := NamespaceName,
		catchPointPOUName := __POUNAME(),
		catchPointPosition := __POSITION()
	);	

	exceptionReaction := OnHandleException(exception := exception, failedMethodName := 'OnBeforeChildrenWorking');

	ProcessException(
		exception := exception,
		exceptionReaction := exceptionReaction,
		exceptionSourceHint := "OnBeforeChildrenWorking error"
	);

	IF exceptionReaction = TOF_Core.EXCEPTION_REACTION.SET_ERROR_AND_STOP THEN
		RETURN;		
	END_IF
__ENDTRY	

IF NOT Enabled OR_ELSE _OperationalState <> OPERATIONAL_STATE.WORKING THEN
	RETURN;
END_IF

FOR i := 0 TO ChildCount - 1 DO
	child := TryGetChildByIndex(index := i);
	
	IF child <> 0
		AND_THEN child.Enabled
		AND_THEN (
			child.OperationalState = OPERATIONAL_STATE.WORKING
			OR_ELSE child.OperationalState = OPERATIONAL_STATE.STOPPED
		)
	THEN
		child.Execute();
		
		IF child.HasError AND_THEN child.Error.Severity = TOF_Core.ERROR_SEVERITY.CRITICAL THEN
			childCriticalErrorReaction := HandleChildCriticalError(childWithError := child);
			
			ProcessChildError(
				childError := child.Error,
				childErrorReaction := childCriticalErrorReaction,
				childErrorSourceHint := TOF_Core.WideStrings.Concat255("Child[", TO_WSTRING(i), "](", child.Name, ").Execute error")
			);
			
			IF childCriticalErrorReaction = CHILD_CRITICAL_ERROR_REACTION.SET_ERROR_AND_STOP THEN
				RETURN;
			END_IF
		END_IF
	END_IF

	IF NOT Enabled OR_ELSE _OperationalState <> OPERATIONAL_STATE.WORKING THEN
		RETURN;
	END_IF
END_FOR

__TRY
	OnAfterChildrenWorking();
__CATCH(exceptionCode)
	exception := TOF_Core.ExceptionManager.GetLastException(
		exceptionCode := exceptionCode,
		catchPointNamespaceName := NamespaceName,
		catchPointPOUName := __POUNAME(),
		catchPointPosition := __POSITION()
	);	

	exceptionReaction := OnHandleException(exception := exception, failedMethodName := 'OnAfterChildrenWorking');

	ProcessException(
		exception := exception,
		exceptionReaction := exceptionReaction,
		exceptionSourceHint := "OnAfterChildrenWorking error"
	);

	IF exceptionReaction = TOF_Core.EXCEPTION_REACTION.SET_ERROR_AND_STOP THEN
		RETURN;		
	END_IF
__ENDTRY
END_METHOD

(*!
<summary>Enables the branch, optionally its children, and invokes enable hooks.</summary>
<description>
Enabling does not automatically reset a STOPPED branch or STOPPED children; they remain STOPPED after
Enable until explicitly Reset. If this branch has a disabled parent, enables the parent with
includeChildren := FALSE.
</description>
<param name="includeChildren">When TRUE, recursively enables child components.</param>
*)
METHOD FINAL Enable
VAR_INPUT
	includeChildren : BOOL := TRUE;
END_VAR
VAR
	i : INT;
	
	child : IChildAutomationComponent;

	exceptionCode : __SYSTEM.ExceptionCode;
	
	thisAsChildAutomationComponent : IChildAutomationComponent;
	parent : IParentAutomationComponent;
END_VAR
VAR_INST
	enabling : BOOL;
END_VAR
IF _Enabled OR_ELSE enabling THEN
	RETURN;
END_IF

enabling := TRUE;

__TRY
	OnBeforeChildrenEnable();
	
	IF includeChildren THEN
		FOR i := 0 TO ChildCount - 1 DO
			child := TryGetChildByIndex(index := i);
			
			IF child <> 0 THEN
				child.Enable(includeChildren := includeChildren);
			END_IF
		END_FOR	
	END_IF
	
	OnAfterChildrenEnable();
	
	IF __QUERYINTERFACE(THIS^, thisAsChildAutomationComponent) THEN
		parent := thisAsChildAutomationComponent.Parent;

		IF parent <> 0 AND_THEN NOT parent.Enabled THEN
			parent.Enable(includeChildren := FALSE);
		END_IF
	END_IF
	
	_Enabled := TRUE;
	
	enabling := FALSE;
__CATCH(exceptionCode)
	enabling := FALSE;
	
	TOF_Core.ExceptionManager.ReThrowLastException(
		exceptionCode := exceptionCode,
		catchPointNamespaceName := NamespaceName,
		catchPointPOUName := __POUNAME(),
		catchPointPosition := __POSITION()
	);
__ENDTRY
END_METHOD

(*!
<summary>Services an initialized branch and advances its enabled execution phases.</summary>
<description>
Only WORKING and STOPPED are serviced. Cycle-service hooks run even while disabled, before and after
enabled input, working or stopped, and output phases. They may enable, disable, stop or reset the branch;
enablement is checked again before work and output. INITIALIZING and INVALID do nothing. The final service
hook also follows handled stop reactions; an escaping nested failure may abort the call. Use one owner task
without recursive Execute. Completed callback effects are not rolled back.
</description>
*)
{attribute 'estimated-stack-usage' := '99'}
METHOD FINAL Execute
VAR
	exceptionCode : __SYSTEM.ExceptionCode;
	exception : TOF_Core.IException;
	exceptionReaction : TOF_Core.EXCEPTION_REACTION;
	runEnabledPhases : BOOL;
END_VAR
IF _OperationalState <> OPERATIONAL_STATE.WORKING
	AND_THEN _OperationalState <> OPERATIONAL_STATE.STOPPED
THEN
	RETURN;
END_IF

runEnabledPhases := TRUE;

__TRY
	OnCycleStart();
__CATCH(exceptionCode)
	exception := TOF_Core.ExceptionManager.GetLastException(
		exceptionCode := exceptionCode,
		catchPointNamespaceName := NamespaceName,
		catchPointPOUName := __POUNAME(),
		catchPointPosition := __POSITION()
	);
	exceptionReaction := OnHandleException(exception := exception, failedMethodName := 'OnCycleStart');

	ProcessException(
		exception := exception,
		exceptionReaction := exceptionReaction,
		exceptionSourceHint := "OnCycleStart error"
	);

	IF exceptionReaction = TOF_Core.EXCEPTION_REACTION.SET_ERROR_AND_STOP THEN
		runEnabledPhases := FALSE;
	END_IF
__ENDTRY

IF runEnabledPhases AND_THEN Enabled THEN
	__TRY
		OnBeforeExecute();
	__CATCH(exceptionCode)
		exception := TOF_Core.ExceptionManager.GetLastException(
			exceptionCode := exceptionCode,
			catchPointNamespaceName := NamespaceName,
			catchPointPOUName := __POUNAME(),
			catchPointPosition := __POSITION()
		);
		exceptionReaction := OnHandleException(exception := exception, failedMethodName := 'OnBeforeExecute');

		ProcessException(
			exception := exception,
			exceptionReaction := exceptionReaction,
			exceptionSourceHint := "OnBeforeExecute error"
		);

		IF exceptionReaction = TOF_Core.EXCEPTION_REACTION.SET_ERROR_AND_STOP THEN
			runEnabledPhases := FALSE;
		END_IF
	__ENDTRY

	IF runEnabledPhases AND_THEN Enabled THEN
		CASE _OperationalState OF
			OPERATIONAL_STATE.WORKING:
				doWork();

			OPERATIONAL_STATE.STOPPED:
				doStop();
		END_CASE
	END_IF

	IF runEnabledPhases AND_THEN Enabled THEN
		__TRY
			OnAfterExecute();
		__CATCH(exceptionCode)
			exception := TOF_Core.ExceptionManager.GetLastException(
				exceptionCode := exceptionCode,
				catchPointNamespaceName := NamespaceName,
				catchPointPOUName := __POUNAME(),
				catchPointPosition := __POSITION()
			);
			exceptionReaction := OnHandleException(exception := exception, failedMethodName := 'OnAfterExecute');

			ProcessException(
				exception := exception,
				exceptionReaction := exceptionReaction,
				exceptionSourceHint := "OnAfterExecute error"
			);
		__ENDTRY
	END_IF
END_IF

__TRY
	OnCycleEnd();
__CATCH(exceptionCode)
	exception := TOF_Core.ExceptionManager.GetLastException(
		exceptionCode := exceptionCode,
		catchPointNamespaceName := NamespaceName,
		catchPointPOUName := __POUNAME(),
		catchPointPosition := __POSITION()
	);
	exceptionReaction := OnHandleException(exception := exception, failedMethodName := 'OnCycleEnd');

	ProcessException(
		exception := exception,
		exceptionReaction := exceptionReaction,
		exceptionSourceHint := "OnCycleEnd error"
	);
__ENDTRY
END_METHOD

METHOD GetEffectiveChildCriticalErrorHandlingPolicy : IChildCriticalErrorHandlingPolicy
VAR
	thisAsChildAutomationComponent : IChildAutomationComponent;
	parent : IParentAutomationComponent;
END_VAR
IF _ChildCriticalErrorHandlingPolicy <> 0 THEN
	GetEffectiveChildCriticalErrorHandlingPolicy := _ChildCriticalErrorHandlingPolicy;
ELSIF __QUERYINTERFACE(THIS^, thisAsChildAutomationComponent) THEN
	parent := thisAsChildAutomationComponent.Parent;

	IF parent <> 0 THEN
		GetEffectiveChildCriticalErrorHandlingPolicy := parent.GetEffectiveChildCriticalErrorHandlingPolicy();
	END_IF
END_IF
END_METHOD

METHOD PROTECTED FINAL HandleChildCriticalError : CHILD_CRITICAL_ERROR_REACTION
VAR_INPUT
	childWithError : IChildAutomationComponent;
END_VAR
VAR
	effectiveChildCriticalErrorHandlingPolicy : IChildCriticalErrorHandlingPolicy;
END_VAR
effectiveChildCriticalErrorHandlingPolicy := GetEffectiveChildCriticalErrorHandlingPolicy();

IF effectiveChildCriticalErrorHandlingPolicy <> 0 THEN
	HandleChildCriticalError := effectiveChildCriticalErrorHandlingPolicy.HandleChildCriticalError(
		childWithError := childWithError,
		handlingObject := THIS^
	);
ELSE
	HandleChildCriticalError := CHILD_CRITICAL_ERROR_REACTION.SET_ERROR_AND_STOP;
END_IF
END_METHOD

(*!
<summary>Checks whether any enabled child still holds a critical error handled with continue.</summary>
<description>
Prevents premature automatic non-critical error clearing and OnRecover calls while an enabled child
remains faulted with a critical error under SET_ERROR_AND_CONTINUE.
</description>
*)
METHOD PRIVATE hasActiveChildCriticalError : BOOL
VAR
	i : INT;
	child : IChildAutomationComponent;
	childCriticalErrorReaction : CHILD_CRITICAL_ERROR_REACTION;
END_VAR
FOR i := 0 TO ChildCount - 1 DO
	child := TryGetChildByIndex(index := i);

	IF child <> 0
		AND_THEN child.Enabled
		AND_THEN child.HasError
		AND_THEN child.Error.Severity = TOF_Core.ERROR_SEVERITY.CRITICAL
	THEN
		childCriticalErrorReaction := HandleChildCriticalError(childWithError := child);

		IF childCriticalErrorReaction = CHILD_CRITICAL_ERROR_REACTION.SET_ERROR_AND_CONTINUE THEN
			hasActiveChildCriticalError := TRUE;

			RETURN;
		END_IF
	END_IF
END_FOR
END_METHOD

(*!
<summary>Validates required dependencies and advances branch initialization.</summary>
<description>
Required storage and child slots are checked before initialization hooks. Empty compositions are valid.
Before the first initialization hook, each child must name this branch as Parent and appear in exactly one slot.
Keep the composition stable thereafter. A mismatch or duplicate records a critical error and makes the branch INVALID.
An INVALID child immediately makes this branch INVALID and copies its error when available.
During initialization, the branch expands its effective initialization timeout to at least the maximum
InitializationTimeout of its children. OnAfterChildrenInitializing runs only once all children have completed
initialization. FALSE reports pending work or failure. Caught initialization failures return FALSE and record
a critical error in terminal INVALID. TRUE reports completed initialization, including an already stopped
component. Callback effects are not rolled back. Child types require a live constructor-bound parent.
</description>
*)
METHOD FINAL Initialize : BOOL
VAR
	i : INT;
	previousIndex : INT;
	expectedParent : IParentAutomationComponent;
	childParent : IParentAutomationComponent;
	hierarchyError : WSTRING(255);
		
	child : IChildAutomationComponent;
	previousChild : IChildAutomationComponent;
	childInitialized : BOOL;
	
	exceptionCode : __SYSTEM.ExceptionCode;
	exception : TOF_Core.IException;
	
END_VAR
IF _OperationalState <> OPERATIONAL_STATE.INITIALIZING THEN
	Initialize := _OperationalState <> OPERATIONAL_STATE.INVALID;

	RETURN;
END_IF

__TRY
	Validate();
	expectedParent := THIS^;

	FOR i := 0 TO ChildCount - 1 DO
		child := TryGetChildByIndex(index := i);

		IF child = 0 THEN
			TOF_Core.Exceptions.ThrowDataMemberNotSpecified(
				sourceNamespaceName := NamespaceName,
				sourceClassName := ClassName,
				sourcePOUName := __POUNAME(),
				sourcePosition := __POSITION(),
				dataMemberName := TOF_Core.Strings.Concat255('Child[', TO_STRING(i), ']')
			);			
		END_IF

		IF _ChildHierarchyValidated THEN
			CONTINUE;
		END_IF

		childParent := child.Parent;

		IF childParent <> expectedParent THEN
			hierarchyError := TOF_Core.WideStrings.Concat255(
				Name,
				": Children[",
				TO_WSTRING(i),
				"] (",
				child.Name,
				") has a different Parent"
			);
		ELSE
			FOR previousIndex := 0 TO i - 1 DO
				previousChild := TryGetChildByIndex(index := previousIndex);

				IF previousChild = child THEN
					hierarchyError := TOF_Core.WideStrings.Concat255(
						Name,
						": Children[",
						TO_WSTRING(i),
						"] (",
						child.Name,
						") duplicates Children[",
						TO_WSTRING(previousIndex),
						"]"
					);

					EXIT;
				END_IF
			END_FOR
		END_IF

		IF hierarchyError <> "" THEN
			TOF_Core.Exceptions.ThrowClassInitialization(
				sourceNamespaceName := NamespaceName,
				sourceClassName := ClassName,
				sourcePOUName := __POUNAME(),
				sourcePosition := __POSITION(),
				errorMessage := hierarchyError
			);
		END_IF
	END_FOR

	_ChildHierarchyValidated := TRUE;
	OnBeforeChildrenInitializing();

	IF _InitializationTimer.PT = T#0S THEN
		_InitializationTimer.PT := Parameters.InitializationTimeout;
	END_IF

	Initialize := TRUE;

	FOR i := 0 TO ChildCount - 1 DO
		child := TryGetChildByIndex(index := i);

		IF child = 0 THEN
			TOF_Core.Exceptions.ThrowDataMemberNotSpecified(
				sourceNamespaceName := NamespaceName,
				sourceClassName := ClassName,
				sourcePOUName := __POUNAME(),
				sourcePosition := __POSITION(),
				dataMemberName := TOF_Core.Strings.Concat255('Child[', TO_STRING(i), ']')
			);
		END_IF

		childInitialized := child.Initialize();

		IF child.OperationalState = OPERATIONAL_STATE.INVALID THEN
			Initialize := FALSE;

			IF child.HasError THEN
				_Error := child.Error;
				_Error.SetSeverity(severity := TOF_Core.ERROR_SEVERITY.CRITICAL);
				SetOperationalState(
					state := OPERATIONAL_STATE.INVALID,
					reason := TOF_Core.WideStrings.Concat255("Child[", TO_WSTRING(i), "] initialization failed")
				);

				RETURN;
			END_IF

			TOF_Core.Exceptions.ThrowStandard(
				sourceNamespaceName := NamespaceName,
				sourceClassName := ClassName,
				sourcePOUName := __POUNAME(),
				sourcePosition := __POSITION(),
				message := "A child entered INVALID during initialization without an error diagnostic."
			);
		END_IF

		IF child.InitializationTimeout > _InitializationTimer.PT THEN
			_InitializationTimer.PT := child.InitializationTimeout;
		END_IF

		Initialize := Initialize AND childInitialized;
	END_FOR

	Initialize := Initialize AND_THEN OnAfterChildrenInitializing();
	
	IF Initialize THEN
		SetOperationalState(state := OPERATIONAL_STATE.WORKING, reason := "Successfull initialization");
	ELSE
		_InitializationTimer(IN := TRUE);
		
		IF _InitializationTimer.Q THEN		
			TOF_Core.Exceptions.ThrowTimeout(
				sourceNamespaceName := NamespaceName,
				sourceClassName := ClassName,
				sourcePOUName := __POUNAME(),
				sourcePosition := __POSITION(),
				timeoutValue := _InitializationTimer.PT,
				operationName := "Initialization"
			);
		END_IF		
	END_IF	
__CATCH(exceptionCode)
	Initialize := FALSE;

	IF hierarchyError = "" THEN
		hierarchyError := "Initialization error";
	END_IF

	exception := TOF_Core.ExceptionManager.GetLastException(
		exceptionCode := exceptionCode,
		catchPointNamespaceName := NamespaceName,
		catchPointPOUName := __POUNAME(),
		catchPointPosition := __POSITION()
	);
	
	ProcessException(
		exception := exception,
		exceptionReaction := TOF_Core.EXCEPTION_REACTION.SET_ERROR_AND_CONTINUE,
		exceptionSourceHint := hierarchyError
	);					
__ENDTRY
END_METHOD

METHOD PROTECTED OnAfterChildrenDisable
END_METHOD

METHOD PROTECTED OnAfterChildrenEnable
END_METHOD

(*!
<summary>Completes branch initialization after all children have finished initializing.</summary>
<description>
Invoked only once every child has completed initialization (returned TRUE from Initialize). Return FALSE to
keep the branch in INITIALIZING until a subsequent Initialize call returns TRUE.
</description>
*)
METHOD PROTECTED OnAfterChildrenInitializing : BOOL
OnAfterChildrenInitializing := TRUE;
END_METHOD

METHOD PROTECTED OnAfterChildrenProcessInput
END_METHOD

(*!
<summary>Runs after the branch completes an output pass without changing its operational state.</summary>
<description>Both working and stopped passes may complete. An interrupted pass skips this hook.</description>
*)
METHOD PROTECTED OnAfterChildrenProcessOutput
END_METHOD

METHOD PROTECTED OnAfterChildrenReset
END_METHOD

METHOD PROTECTED OnAfterChildrenStopped
END_METHOD

METHOD PROTECTED OnAfterChildrenWorking
END_METHOD

(*!
<summary>Completes enabled processing after the working or stopped phase.</summary>
<description>
Execute checks Enabled again before calling this hook. STOPPED branches remain eligible. A handled stop
reaction in OnCycleStart or OnBeforeExecute skips this hook. The base implementation does nothing.
Exceptions follow the branch exception policy.
</description>
*)
METHOD PROTECTED OnAfterExecute
END_METHOD

METHOD PROTECTED OnBeforeChildrenDisable
END_METHOD

METHOD PROTECTED OnBeforeChildrenEnable
END_METHOD

(*!
<summary>Runs before child initialization on each pending initialization cycle.</summary>
<description>
Invoked after branch dependencies and child hierarchy validation succeed. Exceptions transition the branch to
terminal INVALID.
</description>
*)
METHOD PROTECTED OnBeforeChildrenInitializing
END_METHOD

METHOD PROTECTED OnBeforeChildrenProcessInput
END_METHOD

METHOD PROTECTED OnBeforeChildrenProcessOutput
END_METHOD

METHOD PROTECTED OnBeforeChildrenReset
END_METHOD

(*!
<summary>Runs before stopped-child traversal.</summary>
<description>
May call Reset. A state or enablement change ends this stopped phase before remaining children
and the after-stopped hook. Do not recursively call Execute.
</description>
*)
METHOD PROTECTED OnBeforeChildrenStopped
END_METHOD

METHOD PROTECTED OnBeforeChildrenWorking
END_METHOD

(*!
<summary>Prepares an enabled branch for its working or stopped phase.</summary>
<description>
Execute calls this hook after OnCycleStart if the branch is enabled and the enabled phases may proceed.
Execute then checks Enabled again and selects the phase using the current operational state. The base
implementation does nothing. Exceptions follow the branch exception policy.
</description>
*)
METHOD PROTECTED OnBeforeExecute
END_METHOD

(*!
<summary>Services the branch after the enabled phases have run or been skipped.</summary>
<description>
Execute reaches this hook even while disabled and after a handled stop reaction. An escaping exception
can end Execute before this hook runs. The base implementation does nothing. Exceptions raised here follow
the branch exception policy.
</description>
*)
METHOD PROTECTED OnCycleEnd
END_METHOD

(*!
<summary>Services the branch before Execute checks Enabled.</summary>
<description>
Execute calls this hook in WORKING and STOPPED, including while disabled. An override can process commands
that enable or disable the branch for this call. The base implementation does nothing. Exceptions follow
the branch exception policy.
</description>
*)
METHOD PROTECTED OnCycleStart
END_METHOD

(*!
<summary>
Checks local permission and then requests permission from the parent, stopping at the first rejection.
</summary>
<description>
A missing local policy permits this level. The local policy receives this branch as evaluatingObject; the
original descriptor and requester are forwarded unchanged to the parent. Returns TRUE only if no level rejects
the request. On FALSE, rejectReason contains the rejecting level's reason; on TRUE it must be ignored.
Evaluation exceptions propagate to the caller without becoming ordinary rejections. Inputs must be non-null
and live. Arguments are borrowed only during this synchronous call, without ownership transfer.
</description>
*)

METHOD FINAL RequestActionPermission : BOOL
VAR_INPUT
	actionDescriptor : TOF_Core.INamed;
	requestingObject : TOF_Core.IObject;
END_VAR
VAR_IN_OUT
	rejectReason : WSTRING(255);
END_VAR
VAR
	thisAsChildAutomationComponent : IChildAutomationComponent;
	parent : IParentAutomationComponent;
END_VAR
IF _ActionPermissionPolicy <> 0 THEN 
	RequestActionPermission := _ActionPermissionPolicy.CheckActionPermission(
		actionDescriptor := actionDescriptor,
		requestingObject := requestingObject,
		evaluatingObject := THIS^,
		rejectReason := rejectReason
	);
ELSE
	RequestActionPermission := TRUE;
END_IF

IF RequestActionPermission
	AND_THEN __QUERYINTERFACE(THIS^, thisAsChildAutomationComponent)
THEN
	parent := thisAsChildAutomationComponent.Parent;

	IF parent <> 0 THEN
		RequestActionPermission := parent.RequestActionPermission(
			actionDescriptor := actionDescriptor,
			requestingObject := requestingObject,
			rejectReason := rejectReason
		);
	END_IF
END_IF
END_METHOD

(*!
<summary>Attempts to resume an enabled stopped branch and its enabled children.</summary>
<description>
Clears the previous branch error before reset hooks. Disabled children are skipped and remain STOPPED if
later enabled until explicitly Reset. A failure of the branch's own reset hook (OnBeforeChildrenReset or
OnAfterChildrenReset) always leaves the branch STOPPED with a copied CRITICAL error without consulting
ExceptionHandlingPolicy; later children are not reset after OnBeforeChildrenReset fails. Ignore and
continue allow later children to reset and the branch to enter WORKING even if a child remains stopped.
Continue copies that error at ERROR severity; ignore leaves it local. Stop leaves the branch STOPPED. Reset
may be called from a stopped-cycle hook, but reset hooks must not reenter Reset. State or enablement changes
end traversal; completed effects remain.
</description>
*)
METHOD FINAL Reset
VAR
	exceptionCode : __SYSTEM.ExceptionCode;
	exception : TOF_Core.IException;	
	
	childCriticalErrorReaction : CHILD_CRITICAL_ERROR_REACTION;
	
	i : INT;
		
	child : IChildAutomationComponent;	
END_VAR
IF NOT Enabled OR_ELSE _OperationalState <> OPERATIONAL_STATE.STOPPED THEN
	RETURN;
END_IF

_Error.Clear();

__TRY
	OnBeforeChildrenReset();
__CATCH(exceptionCode)		
	exception := TOF_Core.ExceptionManager.GetLastException(
		exceptionCode := exceptionCode,
		catchPointNamespaceName := NamespaceName,
		catchPointPOUName := __POUNAME(),
		catchPointPosition := __POSITION()
	);

	// A failed reset hook always keeps the branch STOPPED with a critical error; the policy is not consulted.
	ProcessException(
		exception := exception,
		exceptionReaction := TOF_Core.EXCEPTION_REACTION.SET_ERROR_AND_STOP,
		exceptionSourceHint := "OnBeforeChildrenReset error"
	);

	RETURN;
__ENDTRY

IF NOT Enabled OR_ELSE _OperationalState <> OPERATIONAL_STATE.STOPPED THEN
	RETURN;
END_IF

FOR i := 0 TO ChildCount - 1 DO
	child := TryGetChildByIndex(index := i);
	
	IF child <> 0 AND_THEN child.Enabled THEN
		child.Reset();
		
		IF child.HasError AND_THEN child.Error.Severity = TOF_Core.ERROR_SEVERITY.CRITICAL THEN
			childCriticalErrorReaction := HandleChildCriticalError(childWithError := child);
			
			ProcessChildError(
				childError := child.Error,
				childErrorReaction := childCriticalErrorReaction,
				childErrorSourceHint := TOF_Core.WideStrings.Concat255("Child[", TO_WSTRING(i), "](", child.Name, ").Reset error")
			);

			IF childCriticalErrorReaction = CHILD_CRITICAL_ERROR_REACTION.SET_ERROR_AND_STOP THEN
				RETURN;
			END_IF
		END_IF
	END_IF

	IF NOT Enabled OR_ELSE _OperationalState <> OPERATIONAL_STATE.STOPPED THEN
		RETURN;
	END_IF
END_FOR

__TRY
	OnAfterChildrenReset();
	
	IF Enabled AND_THEN _OperationalState = OPERATIONAL_STATE.STOPPED THEN
		SetOperationalState(state := OPERATIONAL_STATE.WORKING, reason := "Reset");
	END_IF
__CATCH(exceptionCode)		
	exception := TOF_Core.ExceptionManager.GetLastException(
		exceptionCode := exceptionCode,
		catchPointNamespaceName := NamespaceName,
		catchPointPOUName := __POUNAME(),
		catchPointPosition := __POSITION()
	);

	// A failed reset hook always keeps the branch STOPPED with a critical error; the policy is not consulted.
	ProcessException(
		exception := exception,
		exceptionReaction := TOF_Core.EXCEPTION_REACTION.SET_ERROR_AND_STOP,
		exceptionSourceHint := "OnAfterChildrenReset error"
	);
__ENDTRY
END_METHOD

(*!
<summary>Transitions a WORKING branch and all WORKING children to OPERATIONAL_STATE.STOPPED.</summary>
<description>
Stops the branch and all WORKING children regardless of Enabled. Child Stop failures are logged as critical.
</description>
<param name="reason">Descriptive reason stored in OperationalStateReason.</param>
*)
METHOD FINAL Stop
VAR_INPUT
	reason : WSTRING(255) := "External stop";
END_VAR
VAR
	exceptionCode : __SYSTEM.ExceptionCode;
	exception : TOF_Core.IException;	

	i : INT;
	
	child : IChildAutomationComponent;
END_VAR
IF _OperationalState <> OPERATIONAL_STATE.WORKING THEN
	RETURN;
END_IF

SetOperationalState(state := OPERATIONAL_STATE.STOPPED, reason := reason);

FOR i := 0 TO ChildCount - 1 DO
	__TRY
		child := TryGetChildByIndex(index := i); 
		
		IF child <> 0 AND_THEN child.OperationalState = OPERATIONAL_STATE.WORKING THEN		
			child.Stop(reason := TOF_Core.WideStrings.Concat255("Parent (", Name, ") stopped. Reason: ", reason));
		END_IF			
	__CATCH(exceptionCode)
		exception := TOF_Core.ExceptionManager.GetLastException(
			exceptionCode := exceptionCode,
			catchPointNamespaceName := NamespaceName,
			catchPointPOUName := __POUNAME(),
			catchPointPosition := __POSITION()
		);	
		
		TOF_Core.LogManager.TryLogException(
			exception := exception,
			severity := TOF_Core.ERROR_SEVERITY.CRITICAL,
			topic1 := "AutomationComponent",
			topic2 := "AutomationComponent.Stop"
		);
	__ENDTRY
END_FOR
END_METHOD

(*!
<summary>Returns a borrowed child by its zero-based index.</summary>
<description>
Returns null when the entry is unavailable, the index is out of range or a nested call raises an exception.
Fatal allocation observations return null and leave the fatal latch set for the outer task boundary.
Does not transfer ownership or extend lifetime. Implementations must not propagate exceptions.
</description>
*)
METHOD ABSTRACT TryGetChildByIndex : IChildAutomationComponent
VAR_INPUT
	index : TOF_Core.INT_INDEX;
END_VAR
END_METHOD

METHOD PROTECTED ABSTRACT Validate
END_METHOD

END_FUNCTION_BLOCK

// ---- AutomationComponent/AutomationComponent.TcPOU
(*
SPDX-FileCopyrightText: © 2026 Oleksandr Tiutyk <trofimich@gmail.com>
SPDX-License-Identifier: MIT
License: https://opensource.org/license/mit
*)

(*!
<summary>Provides common automation state, diagnostics and local event reception.</summary>
<description>
Both event delivery directions call OnEventReceived locally. Descendants with a parent or children extend the
appropriate direction with forwarding; terminal nodes only receive the event. Event delivery is synchronous
and borrowed, without retaining the event or transferring ownership. Delivery and forwarding are independent
of Enabled and operational state. OnEventReceived decides whether the component should react in its current
state; inactivity alone does not stop propagation. The event must be non-null and live. Handler exceptions
abort delivery and propagate to the caller; effects of handlers already invoked are not rolled back.
Initialization validates required dependencies before hooks. Child types require a live borrowed parent.
FALSE reports pending initialization or failure; INVALID must never report successful initialization.
Error and HasError observe the same diagnostic selected by GetReportedError(). The base exposes its execution error.
Required error snapshots precede logging callbacks so they preserve the primary diagnostic.
Stop transitions a WORKING component (and, for branches, all WORKING children) to STOPPED regardless of
Enabled, so a runtime stop reaction also stops a disabled working component and preserves its Reset requirement.
</description>
*)

FUNCTION_BLOCK ABSTRACT AutomationComponent EXTENDS TOF_Core.Object IMPLEMENTS IAutomationComponent
VAR
	{attribute 'hide'} 
	_Name : WSTRING;

	{attribute 'hide'} 
	_Enabled : BOOL := TRUE;
	
	{attribute 'hide'} 
	_OperationalState : OPERATIONAL_STATE;
	//! <summary>Counts state transitions so output traversal can detect a stop followed by an immediate reset.</summary>
	_OperationalStateRevision : UDINT;	
	{attribute 'hide'} 
	_OperationalStateReason : WSTRING(255);	

	_InitializationTimer : Tc2_Standard.TON;
	
	{attribute 'hide'} 
	_Error : TOF_Core.ERROR;
	
	{attribute 'hide'} 
	_ExceptionHandlingPolicy : TOF_Core.IExceptionHandlingPolicy;
END_VAR

(*!
<summary>Receives a broadcast event locally without forwarding it.</summary>
<description>
Calls OnEventReceived once. This is the terminal behavior for a leaf; branches override it to forward to
children unless propagation is stopped. Handled does not suppress delivery. The event is borrowed for this
synchronous call and is not retained or owned by the component.
</description>
*)

METHOD BroadcastEvent
VAR_INPUT
	event : TOF_Core.IEvent;
END_VAR
VAR
	stopPropagation : BOOL;
END_VAR
OnEventReceived(event := event, stopPropagation => stopPropagation);
END_METHOD

(*!
<summary>Receives a bubbling event locally without forwarding it.</summary>
<description>
Calls OnEventReceived once. This is the terminal behavior for a root; components with a parent override it to
forward upward unless propagation is stopped. Handled does not suppress delivery. The event is borrowed for
this synchronous call and is not retained or owned by the component.
</description>
*)

METHOD BubbleEvent
VAR_INPUT
	event : TOF_Core.IEvent;
END_VAR
VAR
	stopPropagation : BOOL;
END_VAR
OnEventReceived(event := event, stopPropagation => stopPropagation);
END_METHOD

(*!
<summary>Disables cyclic execution and invokes disable hooks.</summary>
<description>
Branches also disable their children. Hook exceptions propagate to the caller without rolling back prior
effects.
</description>
*)
METHOD ABSTRACT Disable
END_METHOD

(*!
<summary>Enables cyclic execution and invokes enable hooks.</summary>
<description>
Enabling does not automatically reset a STOPPED component; components stopped while disabled or disabled
while stopped remain STOPPED after Enable until explicitly Reset.
</description>
<param name="includeChildren">When TRUE on a branch, recursively enables child components.</param>
*)
METHOD ABSTRACT Enable
VAR_INPUT
	includeChildren : BOOL := TRUE;
END_VAR
END_METHOD

{attribute 'monitoring' := 'call'}
PROPERTY FINAL Enabled : BOOL
GET
Enabled := _Enabled;
END_GET
END_PROPERTY

(*!
<summary>Gets a borrowed view of the currently reported diagnostic.</summary>
<description>
Read the property again after component execution because a descendant can select a different record.
Observe the reference on the owning task while the component is live, following the IErrorProvider contract.
</description>
*)
{attribute 'monitoring' := 'call'}
PROPERTY FINAL Error : REFERENCE TO TOF_Core.ERROR
GET
Error REF= GetReportedError();
END_GET
END_PROPERTY

{attribute 'monitoring' := 'call'}
PROPERTY FINAL ExceptionHandlingPolicy : TOF_Core.IExceptionHandlingPolicy
GET
ExceptionHandlingPolicy := _ExceptionHandlingPolicy;
END_GET
SET
_ExceptionHandlingPolicy := ExceptionHandlingPolicy;
END_SET
END_PROPERTY

METHOD ABSTRACT Execute
END_METHOD

METHOD FB_init : BOOL
VAR_INPUT
	bInitRetains : BOOL; // TRUE: the retain variables are initialized (reset warm / reset cold)
	bInCopyCode : BOOL;  // TRUE: the instance will be copied to the copy code afterward (online change)
	name : WSTRING;
END_VAR
_Name := SEL(
	TOF_Core.WideStrings.IsNullOrWhiteSpace(stringToCheck := name),
	name,
	GetDefaultName()
);
_InitializationTimer.PT := Parameters.InitializationTimeout;
END_METHOD

METHOD FINAL GetEffectiveExceptionHandlingPolicy : TOF_Core.IExceptionHandlingPolicy
VAR
	thisAsChildAutomationComponent : IChildAutomationComponent;
	parent : IParentAutomationComponent;
END_VAR
IF _ExceptionHandlingPolicy <> 0 THEN
	GetEffectiveExceptionHandlingPolicy := _ExceptionHandlingPolicy;
ELSIF __QUERYINTERFACE(THIS^, thisAsChildAutomationComponent) THEN
	parent := thisAsChildAutomationComponent.Parent;

	IF parent <> 0 THEN
		GetEffectiveExceptionHandlingPolicy := parent.GetEffectiveExceptionHandlingPolicy();
	END_IF
END_IF
END_METHOD

METHOD PROTECTED FINAL GetErrorSeverityByExceptionReaction : TOF_Core.ERROR_SEVERITY
VAR_INPUT
	exceptionReaction : TOF_Core.EXCEPTION_REACTION;
END_VAR
IF exceptionReaction = TOF_Core.EXCEPTION_REACTION.SET_ERROR_AND_STOP THEN
	GetErrorSeverityByExceptionReaction := TOF_Core.ERROR_SEVERITY.CRITICAL;
ELSE
	GetErrorSeverityByExceptionReaction := TOF_Core.ERROR_SEVERITY.ERROR;
END_IF
END_METHOD

(*!
<summary>Prepares diagnostic text locally before passing it to read-only logging or exception parameters.</summary>
<description>Computed diagnostic strings are held in local buffers for the duration of the receiving call.</description>
*)
METHOD HandleRequest
VAR_INPUT
	request	: TOF_Core.INamed;
END_VAR
VAR
	formattedLogMessage : TOF_Core.ERROR_MESSAGE;
END_VAR
IF request = 0 THEN
	RETURN;
END_IF

formattedLogMessage := TOF_Core.WideStrings.Concat255("Request ", request.Name, " was not handled");

TOF_Core.LogManager.TryLogMessage(
	message := formattedLogMessage,
	category := TOF_Core.LOG_CATEGORY.INFORMATION,
	topic1 := TO_WSTRING(ClassName),
	topic2 := TO_WSTRING(__POUNAME())
);
END_METHOD

(*!
<summary>Selects the live diagnostic record exposed by Error and HasError.</summary>
<description>
Returns the component's execution record by default. An override must return a valid reference to
instance-owned storage, including when no error is active. Selection must be side-effect free and must
complete without exceptions. Read the selected record on the component's owner task.
</description>
*)
METHOD PROTECTED GetReportedError : REFERENCE TO TOF_Core.ERROR
GetReportedError REF= _Error;
END_METHOD

(*!
<summary>Reports whether the currently selected diagnostic contains an active error.</summary>
*)
{attribute 'monitoring' := 'call'}
PROPERTY FINAL HasError : BOOL
GET
HasError := THIS^.Error.HasError;
END_GET
END_PROPERTY

(*!
<summary>Sets the maximum wait for pending initialization.</summary>
<description>
T#0S selects Parameters.InitializationTimeout immediately upon assignment, so the getter always returns the
active non-zero duration. Branches expand this duration to at least the maximum InitializationTimeout of their
children during initialization.
</description>
*)
{attribute 'monitoring' := 'call'}
PROPERTY FINAL InitializationTimeout : TIME
GET
InitializationTimeout := _InitializationTimer.PT;
END_GET
SET
_InitializationTimer.PT := SEL(
	InitializationTimeout = T#0S,
	InitializationTimeout,
	Parameters.InitializationTimeout
);
END_SET
END_PROPERTY

(*!
<summary>Validates mandatory dependencies and advances initialization.</summary>
<description>
FALSE reports pending work or failure. An INVALID component must never report TRUE. Caught failures
record a critical copied error and enter terminal INVALID. Completed callback effects are not rolled back.
Only a pending call evaluates the timeout. Completion on the deadline cycle succeeds.
</description>
*)
METHOD ABSTRACT Initialize : BOOL
END_METHOD

{attribute 'monitoring' := 'call'}
PROPERTY FINAL Name : REFERENCE TO WSTRING
GET
Name REF= _Name;
END_GET
END_PROPERTY

(*!
<summary>Handles a delivered event locally and can stop further propagation along the current route.</summary>
<description>
May be called regardless of Enabled or operational state, including while disabled or stopped. The handler
checks state when its reaction requires it. Ignoring an event does not stop propagation; leave stopPropagation
FALSE unless further delivery along the route must be stopped. The event must be non-null and live and is
borrowed only for the call; do not retain it for later use. Handled and stopPropagation are independent.
Setting stopPropagation stops bubbling to the parent or broadcasting into this node's descendants; it does not
cancel sibling branches in the caller. An exception aborts delivery and propagates to the dispatch caller,
without rolling back prior effects.
</description>
*)

METHOD OnEventReceived
VAR_INPUT
	event : TOF_Core.IEvent;
END_VAR
VAR_OUTPUT
	stopPropagation : BOOL;
END_VAR
END_METHOD

METHOD PROTECTED FINAL OnHandleException : TOF_Core.EXCEPTION_REACTION
VAR_INPUT
	exception : TOF_Core.IException;
	failedMethodName : STRING(255);
END_VAR
VAR
	effectiveExceptionHandlingPolicy : TOF_Core.IExceptionHandlingPolicy;
END_VAR
effectiveExceptionHandlingPolicy := GetEffectiveExceptionHandlingPolicy();

IF effectiveExceptionHandlingPolicy <> 0 THEN
	OnHandleException := effectiveExceptionHandlingPolicy.HandleException(
		exception := exception,
		handlingObject := THIS^,
		failedMethodName := failedMethodName
	);
ELSE
	OnHandleException := TOF_Core.EXCEPTION_REACTION.SET_ERROR_AND_STOP;
END_IF
END_METHOD

METHOD PROTECTED OnOperationalStateChanged
VAR_INPUT
	previousState : OPERATIONAL_STATE;
END_VAR
END_METHOD

(*!
<summary>Runs at the start of cyclic working execution when clearing a non-critical error.</summary>
<description>
The base implementation does nothing. An exception raised by OnRecover always records a copied CRITICAL
error and stops the component without consulting ExceptionHandlingPolicy.
</description>
*)
METHOD PROTECTED OnRecover
END_METHOD

{attribute 'monitoring' := 'call'}
PROPERTY FINAL OperationalState : OPERATIONAL_STATE
GET
OperationalState := _OperationalState;
END_GET
END_PROPERTY

{attribute 'monitoring' := 'call'}
PROPERTY FINAL OperationalStateReason : REFERENCE TO WSTRING(255)
GET
OperationalStateReason REF= _OperationalStateReason;
END_GET
END_PROPERTY

METHOD PROTECTED ProcessChildError
VAR_INPUT
	childError : REFERENCE TO TOF_Core.ERROR;  
	childErrorReaction : CHILD_CRITICAL_ERROR_REACTION;	
	childErrorSourceHint : WSTRING(255);
END_VAR

IF NOT __ISVALIDREF(childError)
	OR_ELSE childError.Empty
	OR_ELSE childError.Severity <> TOF_Core.ERROR_SEVERITY.CRITICAL
THEN
	RETURN;
END_IF

IF OperationalState <> OPERATIONAL_STATE.INITIALIZING THEN
	CASE childErrorReaction OF
		CHILD_CRITICAL_ERROR_REACTION.SET_ERROR_AND_CONTINUE:
			IF _Error.Empty THEN
				_Error := childError;
				_Error.SetSeverity(severity := TOF_Core.ERROR_SEVERITY.ERROR);
			END_IF		
		
		CHILD_CRITICAL_ERROR_REACTION.SET_ERROR_AND_STOP:
			IF _Error.Empty OR_ELSE _Error.Severity < TOF_Core.ERROR_SEVERITY.CRITICAL THEN
				_Error := childError;
				_Error.SetSeverity(severity := TOF_Core.ERROR_SEVERITY.CRITICAL);
			END_IF	
			
			IF OperationalState = OPERATIONAL_STATE.WORKING THEN
				Stop(reason := childErrorSourceHint);		
			END_IF
	END_CASE
ELSE
	_Error := childError;
	
	SetOperationalState(state := OPERATIONAL_STATE.INVALID, reason := childErrorSourceHint);		
END_IF
END_METHOD

(*!
<summary>Applies an exception reaction to copied diagnostics and operational state.</summary>
<description>
Initialization failures enter INVALID with a critical error. At runtime a stop reaction records a
critical error and calls Stop on a working component, including when disabled (since Stop transitions
WORKING components and WORKING children to STOPPED regardless of Enabled). This preserves the Reset
requirement after a failed disabled service callback. When the reaction requires an error copy, it is
completed before logging callbacks can reuse a task-local exception. Conversion failures may propagate before
logging and state transitions.
</description>
*)
METHOD PROTECTED ProcessException
VAR_INPUT
	exception : TOF_Core.IException;  
	exceptionReaction : TOF_Core.EXCEPTION_REACTION;	
	exceptionSourceHint : WSTRING(255);
END_VAR
IF exception = 0 OR_ELSE exception.Empty THEN
	RETURN;
END_IF

IF OperationalState = OPERATIONAL_STATE.INITIALIZING THEN
	exception.ToError(targetError := _Error, severity := TOF_Core.ERROR_SEVERITY.CRITICAL);
	TOF_Core.LogManager.TryLogException(exception := exception, severity := TOF_Core.ERROR_SEVERITY.CRITICAL);
	SetOperationalState(state := OPERATIONAL_STATE.INVALID, reason := exceptionSourceHint);

	RETURN;
END_IF

CASE exceptionReaction OF
	TOF_Core.EXCEPTION_REACTION.SET_ERROR_AND_CONTINUE:
		IF _Error.Empty THEN
			exception.ToError(targetError := _Error, severity := TOF_Core.ERROR_SEVERITY.ERROR);
		END_IF

	TOF_Core.EXCEPTION_REACTION.SET_ERROR_AND_STOP:
		IF _Error.Empty OR_ELSE _Error.Severity < TOF_Core.ERROR_SEVERITY.CRITICAL THEN
			exception.ToError(targetError := _Error, severity := TOF_Core.ERROR_SEVERITY.CRITICAL);
		END_IF
END_CASE

TOF_Core.LogManager.TryLogException(
	exception := exception,
	severity := GetErrorSeverityByExceptionReaction(exceptionReaction := exceptionReaction)
);

IF exceptionReaction = TOF_Core.EXCEPTION_REACTION.SET_ERROR_AND_STOP
	AND_THEN OperationalState = OPERATIONAL_STATE.WORKING
THEN
	Stop(reason := exceptionSourceHint);
END_IF
END_METHOD

(*!
<summary>Attempts to recover an enabled stopped component to WORKING.</summary>
<description>
Served only while Enabled and STOPPED. Clears the previous error before reset hooks. A failure in the
component's own reset hook always leaves the component STOPPED with a copied CRITICAL error without
consulting ExceptionHandlingPolicy.
</description>
*)
METHOD ABSTRACT Reset
END_METHOD

(*!
<summary>Records the state and reason and notifies descendants on a transition.</summary>
<description>Advances the transition counter before callbacks so an interrupted output pass can be detected.</description>
<param name="state">New operational state.</param>
<param name="reason">Reason recorded even when the state stays the same.</param>
*)
METHOD PROTECTED SetOperationalState
VAR_INPUT
	state : OPERATIONAL_STATE;
	reason : WSTRING(255);
END_VAR
VAR
	previousState : OPERATIONAL_STATE;

	exceptionCode : __SYSTEM.ExceptionCode;
	exception : TOF_Core.IException;
END_VAR
_OperationalStateReason := reason;

IF _OperationalState = state THEN
	RETURN;
END_IF

previousState := _OperationalState;

_OperationalState := state;
_OperationalStateRevision := _OperationalStateRevision + 1;

__TRY
	OnOperationalStateChanged(previousState := previousState);
__CATCH(exceptionCode)
	exception := TOF_Core.ExceptionManager.GetLastException(
		exceptionCode := exceptionCode,
		catchPointNamespaceName := NamespaceName,
		catchPointPOUName := __POUNAME(),
		catchPointPosition := __POSITION()
	);

	TOF_Core.LogManager.TryLogException(
		exception := exception,
		severity := TOF_Core.ERROR_SEVERITY.ERROR,
		topic1 := "AutomationComponent",
		topic2 := "AutomationComponent.OnOperationalStateChanged"
	);
__ENDTRY
END_METHOD

(*!
<summary>Transitions a WORKING component to OPERATIONAL_STATE.STOPPED.</summary>
<description>
Transitions a WORKING component (and, for branches, all WORKING children) to OPERATIONAL_STATE.STOPPED
regardless of Enabled.
</description>
<param name="reason">Descriptive reason stored in OperationalStateReason.</param>
*)
METHOD ABSTRACT Stop
VAR_INPUT
	reason : WSTRING(255) := "External stop";
END_VAR
END_METHOD

END_FUNCTION_BLOCK

// ---- AutomationComponent/Branches/AutomationController/AutomationControllers.TcPOU
(*
SPDX-FileCopyrightText: Â© 2026 Oleksandr Tiutyk <trofimich@gmail.com>
SPDX-License-Identifier: MIT
License: https://opensource.org/license/mit
*)

(*!
<summary>Provides shared constants and metadata for automation controllers.</summary>
<description>
Supplies NoPlugins sentinel array for initializing controllers without extension plugins.
</description>
*)

{attribute 'no_explicit_call' := 'do not call this function block directly'}
PROGRAM AutomationControllers
VAR_OUTPUT CONSTANT
	(*! <summary>Empty array sentinel representing the absence of controller plugins.</summary> *)
	NoPlugins : ARRAY [0..-1] OF IAutomationControllerPlugin := [];
END_VAR
VAR
	_ClassName : STRING := __POUNAME();
END_VAR

(*!
<summary>Gets the class name of the program.</summary>
*)
{attribute 'monitoring' := 'call'}
PROPERTY ClassName : REFERENCE TO STRING
GET
ClassName REF= _ClassName;
END_GET
END_PROPERTY

(*!
<summary>Gets the namespace of the program.</summary>
*)
{attribute 'monitoring' := 'call'}
PROPERTY NamespaceName : REFERENCE TO STRING
GET
NamespaceName REF= CurrentNamespace.Name;
END_GET
END_PROPERTY

END_PROGRAM

// ---- Internal/CurrentNamespace.TcPOU
(*
SPDX-FileCopyrightText: Â© 2026 Oleksandr Tiutyk <trofimich@gmail.com>
SPDX-License-Identifier: MIT
License: https://opensource.org/license/mit
*)

(*!
<summary>Internal helper program providing access to the current library namespace.</summary>
*)

{attribute 'no_explicit_call' := 'do not call this POU directly'}
PROGRAM INTERNAL CurrentNamespace
VAR
	{attribute 'hide'} 
	_NamespaceExtractor : NamespaceExtractor;
END_VAR

(*!
<summary>Gets a reference to the current library namespace string.</summary>
*)
{attribute 'monitoring' := 'call'}
PROPERTY Name : REFERENCE TO STRING
GET
Name REF= _NamespaceExtractor.CurrentNamespace;
END_GET
END_PROPERTY

END_PROGRAM

// ---- Internal/NamespaceExtractor.TcPOU
(*
SPDX-FileCopyrightText: Â© 2026 Oleksandr Tiutyk <trofimich@gmail.com>
SPDX-License-Identifier: MIT
License: https://opensource.org/license/mit
*)

(*!
<summary>Internal helper function block extracting library namespace via attribute init_namespace.</summary>
*)

FUNCTION_BLOCK INTERNAL NamespaceExtractor
VAR_OUTPUT
	{attribute 'init_namespace'} 
	CurrentNamespace : STRING; 	
END_VAR

END_FUNCTION_BLOCK

// ---- AutomationComponent/Branches/AutomationController/Plugins/HMI/HmiAutomationComponentElement.TcPOU
(*
SPDX-FileCopyrightText: © 2026 Oleksandr Tiutyk <trofimich@gmail.com>
SPDX-License-Identifier: MIT
License: https://opensource.org/license/mit
*)

(*!
<summary>Exchanges commands and status between an HMI and an automation component.</summary>
<description>
Derived elements supply component identity and invoke the protected update methods. Error timestamps are reset
to the epoch when no error is reported. Commands received in AutomationComponentCommands are consumed and reset
within the element instance upon dispatch. External HMI systems must write directly to the element's
AutomationComponentCommands symbol or read back the reset state for command handshake.
</description>
*)

FUNCTION_BLOCK ABSTRACT HmiAutomationComponentElement
VAR_INPUT
	AutomationComponentCommands : HMI_AUTOMATION_COMPONENT_COMMANDS;
END_VAR
VAR_OUTPUT
	AutomationComponentStatuses : HMI_AUTOMATION_COMPONENT_STATUSES;
END_VAR

(*!
<summary>Gets the class name of the concrete HMI element.</summary>
*)
{attribute 'monitoring' := 'call'}
PROPERTY ABSTRACT ClassName : REFERENCE TO STRING
GET
END_GET
END_PROPERTY

(*!
<summary>Gets the namespace of the concrete HMI element.</summary>
*)
{attribute 'monitoring' := 'call'}
PROPERTY ABSTRACT NamespaceName : REFERENCE TO STRING
GET
END_GET
END_PROPERTY

(*!
<summary>Dispatches pending HMI commands to the target automation component.</summary>
<description>
Captures and resets the command flags in AutomationComponentCommands to FALSE before invoking Enable,
Disable, or Reset on the target component, preventing repeated execution across cycles if a hook raises an
exception. When both Disable and Enable are set simultaneously, Disable takes precedence. A null component
reference causes an immediate return without mutating commands. External HMI systems must write directly to
the element's AutomationComponentCommands symbol or read back the reset state for command handshake.
</description>
<param name="automationComponent">Target component receiving the dispatched commands.</param>
*)
METHOD PROTECTED ProcessAutomationComponentCommands
VAR_INPUT
	automationComponent : IAutomationComponent;
END_VAR
VAR
	disableRequested : BOOL;
	enableRequested : BOOL;
	resetRequested : BOOL;
END_VAR
IF automationComponent = 0 THEN
	RETURN;
END_IF

disableRequested := AutomationComponentCommands.Disable;
enableRequested := AutomationComponentCommands.Enable;
resetRequested := AutomationComponentCommands.Reset;

AutomationComponentCommands.Disable := FALSE;
AutomationComponentCommands.Enable := FALSE;
AutomationComponentCommands.Reset := FALSE;

IF disableRequested THEN
	automationComponent.Disable();
ELSIF enableRequested THEN
	automationComponent.Enable(includeChildren := TRUE);
END_IF

IF resetRequested THEN
	automationComponent.Reset();
END_IF
END_METHOD

(*!
<summary>Copies current component status to the HMI outputs.</summary>
<description>
A null component leaves outputs unchanged. When no error is reported, clears error text and resets error
timestamps to LongDateAndTimes.EPOCH.
</description>
*)
METHOD PROTECTED UpdateAutomationComponentStatuses
VAR_INPUT
	automationComponent : IAutomationComponent;
END_VAR
IF automationComponent = 0 THEN
	RETURN;
END_IF

AutomationComponentStatuses.Enabled := automationComponent.Enabled;

AutomationComponentStatuses.HasError := automationComponent.HasError;

IF automationComponent.HasError THEN
	AutomationComponentStatuses.ErrorMessage := automationComponent.Error.ToString(
		sourceDisplayMode := TOF_Core.ERROR_SOURCE_DISPLAY_MODE.HIDDEN,
		timestampDisplayMode := TOF_Core.TIMESTAMP_DISPLAY_MODE.HIDDEN
	);
	AutomationComponentStatuses.ErrorSource := automationComponent.Error.GetSource(appendRootSource := TRUE);	
	AutomationComponentStatuses.ErrorLocalTimestamp := automationComponent.Error.LocalTimestamp;
	AutomationComponentStatuses.ErrorUtcTimestamp := automationComponent.Error.UtcTimestamp;
ELSE
	AutomationComponentStatuses.ErrorMessage := "";
	AutomationComponentStatuses.ErrorSource := '';	
	AutomationComponentStatuses.ErrorLocalTimestamp := TOF_Core.LongDateAndTimes.EPOCH;
	AutomationComponentStatuses.ErrorUtcTimestamp := TOF_Core.LongDateAndTimes.EPOCH;
END_IF

AutomationComponentStatuses.OperationalState := automationComponent.OperationalState;
AutomationComponentStatuses.OperationalStateName := TO_STRING(AutomationComponentStatuses.OperationalState);
AutomationComponentStatuses.OperationalStateReason := automationComponent.OperationalStateReason;
END_METHOD

END_FUNCTION_BLOCK

// ---- AutomationComponent/Branches/Composite/CompositeAutomationComponent.TcPOU
(*
SPDX-FileCopyrightText: © 2026 Oleksandr Tiutyk <trofimich@gmail.com>
SPDX-License-Identifier: MIT
License: https://opensource.org/license/mit
*)

(*!
<summary>Provides automation components with indexed access to their related objects.</summary>
<description>
Indexed Try lookups borrow interfaces and contain exceptions. Fatal allocation observations return null
without clearing the latch.
A state transition during output processing skips remaining outputs and the after-output hook.
Completed writes remain effective. A pass started in STOPPED proceeds while the branch stays in that state.
Parent is mandatory and borrowed for the component lifetime.
</description>
*)

FUNCTION_BLOCK ABSTRACT CompositeAutomationComponent
VAR_GENERIC CONSTANT
	{attribute 'hide'} 
    _ChildCount : TOF_Core.INT_LENGTH := 0;
END_VAR
EXTENDS BranchAutomationComponent IMPLEMENTS ICompositeAutomationComponent
VAR
	{attribute 'hide'} 
	_Parent : IParentAutomationComponent;
END_VAR

METHOD FINAL BubbleEvent
VAR_INPUT
	event : TOF_Core.IEvent;
END_VAR
VAR
	stopPropagation : BOOL;
	
	parentAsBubbleEventDispatcher : TOF_Core.IBubbleEventDispatcher;
END_VAR
OnEventReceived(event := event, stopPropagation => stopPropagation);

IF stopPropagation THEN
	RETURN;
END_IF

IF __QUERYINTERFACE(Parent, parentAsBubbleEventDispatcher) THEN
	parentAsBubbleEventDispatcher.BubbleEvent(event := event);
END_IF
END_METHOD

{attribute 'monitoring' := 'call'}
PROPERTY FINAL ChildCount : TOF_Core.INT_LENGTH
GET
ChildCount := _ChildCount;
END_GET
END_PROPERTY

{attribute 'monitoring' := 'call'}
PROPERTY ABSTRACT Children : REFERENCE TO ARRAY [0.._ChildCount - 1] OF IChildAutomationComponent
GET
END_GET
END_PROPERTY

METHOD FB_init : BOOL
VAR_INPUT
	bInitRetains : BOOL; // TRUE: the retain variables are initialized (reset warm / reset cold)
	bInCopyCode : BOOL;  // TRUE: the instance will be copied to the copy code afterward (online change)
	name : WSTRING;
	parent : IParentAutomationComponent;
END_VAR
_Parent := parent;
END_METHOD

(*!
<summary>Borrows the constructor-bound parent for the composite lifetime.</summary>
<description>
The parent is mandatory for initialization and must remain live. Ownership is not transferred.
</description>
*)
{attribute 'monitoring' := 'call'}
PROPERTY FINAL Parent : IParentAutomationComponent
GET
Parent := _Parent;
END_GET
END_PROPERTY

(*!
<summary>Processes enabled input children in slot order.</summary>
<description>
While the branch remains enabled, a transition to STOPPED continues the input pass through the remaining
enabled input children and the after-input hook. Input callbacks must support execution in STOPPED.
</description>
*)
METHOD FINAL ProcessInput
VAR
	exceptionCode : __SYSTEM.ExceptionCode;
	exception : TOF_Core.IException;	
	exceptionReaction : TOF_Core.EXCEPTION_REACTION;
	
